C09149=1146.560,-113.783,-43.527,178.648,5.974,149.471
C09150=1146.565,-114.032,-43.519,178.646,5.974,149.471
C09151=1146.571,-114.282,-43.510,178.644,5.974,149.472
C09152=1146.576,-114.532,-43.501,178.642,5.973,149.472
C09153=1146.581,-114.781,-43.492,178.640,5.973,149.473
C09154=1146.587,-115.031,-43.484,178.638,5.973,149.473
C09155=1146.592,-115.281,-43.475,178.636,5.973,149.474
C09156=1146.598,-115.531,-43.466,178.634,5.972,149.474
C09157=1146.603,-115.781,-43.457,178.632,5.971,149.475
C09158=1146.609,-116.030,-43.449,178.630,5.971,149.475
C09159=1146.614,-116.280,-43.441,178.628,5.970,149.476
C09160=1146.619,-116.530,-43.432,178.627,5.970,149.476
C09161=1146.625,-116.779,-43.424,178.624,5.970,149.477
C09162=1146.630,-117.029,-43.415,178.622,5.970,149.477
C09163=1146.635,-117.279,-43.406,178.620,5.969,149.478
C09164=1146.641,-117.530,-43.398,178.619,5.969,149.478
C09165=1146.646,-117.779,-43.389,178.616,5.969,149.479
C09166=1146.651,-118.028,-43.380,178.614,5.968,149.479
C09167=1146.657,-118.278,-43.371,178.613,5.968,149.480
C09168=1146.663,-118.528,-43.363,178.610,5.967,149.480
C09169=1146.668,-118.778,-43.354,178.609,5.967,149.481
C09170=1146.673,-119.028,-43.346,178.607,5.967,149.481
C09171=1146.678,-119.278,-43.337,178.605,5.967,149.482
C09172=1146.684,-119.527,-43.329,178.602,5.966,149.482
C09173=1146.689,-119.777,-43.320,178.601,5.966,149.483
C09174=1146.695,-120.027,-43.311,178.599,5.966,149.483
C09175=1146.701,-120.277,-43.303,178.597,5.966,149.484
C09176=1146.706,-120.527,-43.294,178.595,5.965,149.484
C09177=1146.710,-120.776,-43.286,178.593,5.965,149.485
C09178=1146.716,-121.026,-43.278,178.591,5.964,149.485
C09179=1146.721,-121.276,-43.269,178.589,5.964,149.486
C09180=1146.727,-121.526,-43.260,178.587,5.963,149.486
C09181=1146.733,-121.776,-43.253,178.585,5.963,149.487
C09182=1146.738,-122.025,-43.244,178.583,5.963,149.487
C09183=1146.743,-122.275,-43.235,178.581,5.962,149.488
C09184=1146.749,-122.525,-43.227,178.579,5.962,149.489
C09185=1146.754,-122.775,-43.219,178.577,5.962,149.489
C09186=1146.759,-123.025,-43.211,178.575,5.962,149.490
C09187=1146.765,-123.274,-43.202,178.573,5.961,149.490
C09188=1146.770,-123.524,-43.193,178.571,5.961,149.491
C09189=1146.775,-123.775,-43.185,178.569,5.960,149.491
C09190=1146.781,-124.024,-43.176,178.568,5.960,149.491
C09191=1146.786,-124.273,-43.168,178.565,5.960,149.492
C09192=1146.791,-124.524,-43.160,178.564,5.960,149.492
C09193=1146.797,-124.773,-43.151,178.562,5.959,149.493
C09194=1146.802,-125.023,-43.143,178.560,5.959,149.493
C09195=1146.808,-125.273,-43.134,178.558,5.958,149.494
C09196=1146.814,-125.523,-43.126,178.556,5.958,149.494
C09197=1146.818,-125.772,-43.118,178.554,5.957,149.495
C09198=1146.824,-126.022,-43.110,178.553,5.957,149.495
C09199=1146.829,-126.272,-43.101,178.550,5.957,149.496
C09200=1146.834,-126.522,-43.093,178.548,5.957,149.497
C09201=1146.840,-126.772,-43.085,178.546,5.956,149.497
C09202=1146.845,-127.021,-43.076,178.544,5.956,149.498
C09203=1146.851,-127.271,-43.069,178.542,5.956,149.498
C09204=1146.856,-127.521,-43.060,178.541,5.956,149.499
C09205=1146.862,-127.771,-43.052,178.538,5.955,149.499
C09206=1146.867,-128.020,-43.043,178.537,5.955,149.500
C09207=1146.872,-128.271,-43.035,178.535,5.954,149.500
C09208=1146.452,-128.281,-43.078,178.531,5.958,149.502
C09209=1146.446,-128.032,-43.087,178.533,5.958,149.501
C09210=1146.441,-127.782,-43.094,178.535,5.959,149.501
C09211=1146.436,-127.532,-43.103,178.537,5.959,149.500
C09212=1146.430,-127.282,-43.111,178.539,5.959,149.500
C09213=1146.425,-127.033,-43.120,178.541,5.959,149.499
C09214=1146.419,-126.783,-43.128,178.543,5.960,149.499
C09215=1146.414,-126.533,-43.136,178.545,5.960,149.498
C09216=1146.409,-126.283,-43.144,178.547,5.961,149.498
C09217=1146.403,-126.034,-43.153,178.549,5.961,149.497
C09218=1146.397,-125.783,-43.161,178.551,5.961,149.497
C09219=1146.392,-125.534,-43.170,178.552,5.961,149.496
C09220=1146.387,-125.284,-43.177,178.555,5.962,149.496
C09221=1146.382,-125.034,-43.186,178.556,5.962,149.495
C09222=1146.376,-124.785,-43.195,178.558,5.963,149.495
C09223=1146.370,-124.534,-43.203,178.560,5.963,149.494
C09224=1146.365,-124.285,-43.212,178.562,5.964,149.494
C09225=1146.360,-124.035,-43.219,178.564,5.964,149.493
C09226=1146.355,-123.785,-43.228,178.566,5.964,149.493
C09227=1146.349,-123.536,-43.236,178.568,5.964,149.492
C09228=1146.344,-123.286,-43.244,178.570,5.965,149.492
C09229=1146.338,-123.036,-43.253,178.571,5.965,149.491
C09230=1146.332,-122.786,-43.261,178.574,5.965,149.491
C09231=1146.327,-122.536,-43.270,178.576,5.965,149.490
C09232=1146.323,-122.287,-43.278,178.578,5.966,149.490
C09233=1146.317,-122.037,-43.286,178.579,5.966,149.489
C09234=1146.311,-121.787,-43.295,178.582,5.967,149.489
C09235=1146.306,-121.537,-43.303,178.583,5.967,149.488
C09236=1146.300,-121.287,-43.312,178.585,5.967,149.488
C09237=1146.295,-121.038,-43.321,178.588,5.968,149.487
C09238=1146.290,-120.787,-43.329,178.589,5.968,149.487
C09239=1146.284,-120.538,-43.337,178.591,5.969,149.486
C09240=1146.279,-120.288,-43.346,178.593,5.969,149.486
C09241=1146.274,-120.039,-43.355,178.595,5.970,149.485
C09242=1146.269,-119.788,-43.363,178.597,5.969,149.485
C09243=1146.263,-119.539,-43.371,178.600,5.970,149.484
C09244=1146.258,-119.289,-43.380,178.601,5.970,149.484
C09245=1146.252,-119.039,-43.388,178.603,5.971,149.483
C09246=1146.247,-118.789,-43.397,178.605,5.971,149.483
C09247=1146.241,-118.540,-43.406,178.607,5.971,149.482
C09248=1146.236,-118.290,-43.415,178.609,5.971,149.482
C09249=1146.230,-118.040,-43.423,178.611,5.972,149.481
C09250=1146.225,-117.790,-43.431,178.613,5.972,149.481
C09251=1146.220,-117.540,-43.440,178.615,5.973,149.480
C09252=1146.214,-117.290,-43.449,178.617,5.973,149.480
C09253=1146.209,-117.041,-43.457,178.619,5.973,149.479
C09254=1146.203,-116.791,-43.466,178.621,5.974,149.478
C09255=1146.198,-116.541,-43.475,178.623,5.974,149.478
C09256=1146.193,-116.291,-43.484,178.625,5.975,149.478
C09257=1146.187,-116.041,-43.492,178.627,5.974,149.477
C09258=1146.182,-115.792,-43.500,178.629,5.975,149.477
C09259=1146.177,-115.542,-43.509,178.630,5.975,149.476
C09260=1146.171,-115.293,-43.518,178.633,5.976,149.476
C09261=1146.166,-115.043,-43.527,178.635,5.977,149.475
C09262=1146.160,-114.792,-43.535,178.637,5.976,149.474
C09263=1146.155,-114.542,-43.544,178.639,5.977,149.474
C09264=1146.149,-114.293,-43.552,178.641,5.977,149.473
C09265=1146.144,-114.043,-43.561,178.643,5.978,149.473
C09266=1146.139,-113.793,-43.570,178.644,5.978,149.472
C09267=1146.134,-113.544,-43.579,178.647,5.978,149.472
C09268=1146.128,-113.294,-43.587,178.648,5.978,149.471
C09269=1146.123,-113.044,-43.596,178.650,5.979,149.471
C09270=1146.117,-112.794,-43.605,178.653,5.980,149.470
C09271=1146.112,-112.544,-43.614,178.655,5.979,149.470
C09272=1146.107,-112.294,-43.623,178.657,5.980,149.469
C09273=1146.101,-112.045,-43.631,178.658,5.980,149.469
C09274=1146.096,-111.795,-43.640,178.661,5.981,149.468
C09275=1146.091,-111.546,-43.649,178.662,5.981,149.468
C09276=1146.086,-111.295,-43.657,178.664,5.982,149.467
C09277=1146.080,-111.045,-43.666,178.667,5.982,149.467
C09278=1146.075,-110.796,-43.674,178.669,5.982,149.466
C09279=1146.069,-110.546,-43.683,178.671,5.983,149.466
C09280=1146.064,-110.296,-43.693,178.673,5.983,149.465
C09281=1146.058,-110.046,-43.702,178.675,5.983,149.465
C09282=1146.053,-109.796,-43.711,178.676,5.983,149.464
C09283=1146.047,-109.547,-43.719,178.679,5.984,149.464
C09284=1146.042,-109.297,-43.728,178.681,5.985,149.463
C09285=1146.037,-109.048,-43.737,178.682,5.985,149.463
C09286=1146.032,-108.798,-43.746,178.685,5.985,149.462
C09287=1146.027,-108.548,-43.755,178.687,5.985,149.462
C09288=1146.022,-108.298,-43.764,178.689,5.986,149.461
C09289=1146.015,-108.049,-43.773,178.691,5.987,149.461
C09290=1146.010,-107.799,-43.782,178.693,5.987,149.460
C09291=1146.005,-107.549,-43.791,178.695,5.987,149.460
C09292=1146.000,-107.299,-43.799,178.697,5.987,149.459
C09293=1145.994,-107.049,-43.808,178.699,5.988,149.458
C09294=1145.989,-106.799,-43.817,178.701,5.988,149.458
C09295=1145.984,-106.550,-43.826,178.703,5.988,149.457
C09296=1145.978,-106.300,-43.835,178.705,5.989,149.457
C09297=1145.972,-106.050,-43.844,178.707,5.989,149.456
C09298=1145.967,-105.800,-43.853,178.709,5.990,149.456
C09299=1145.962,-105.550,-43.862,178.711,5.989,149.455
C09300=1145.957,-105.301,-43.871,178.713,5.990,149.455
C09301=1145.952,-105.051,-43.880,178.715,5.991,149.454
C09302=1145.946,-104.801,-43.889,178.717,5.991,149.454
C09303=1145.940,-104.551,-43.898,178.719,5.992,149.453
C09304=1145.935,-104.302,-43.907,178.721,5.992,149.453
C09305=1145.930,-104.052,-43.916,178.723,5.992,149.452
C09306=1145.925,-103.802,-43.925,178.726,5.993,149.452
C09307=1145.919,-103.552,-43.935,178.727,5.993,149.451
C09308=1145.914,-103.302,-43.944,178.729,5.993,149.451
C09309=1145.908,-103.030,-43.953,178.732,5.994,149.450
C09310=1145.903,-102.758,-43.963,178.734,5.994,149.449
C09311=1145.896,-102.487,-43.973,178.736,5.995,149.449
C09312=1145.891,-102.214,-43.983,178.739,5.995,149.448
C09313=1145.886,-101.964,-43.992,178.741,5.996,149.448
C09314=1145.880,-101.714,-44.001,178.742,5.996,149.447
C09315=1145.875,-101.465,-44.011,178.745,5.996,149.447
C09316=1145.870,-101.215,-44.020,178.746,5.996,149.446
C09317=1145.864,-100.965,-44.029,178.749,5.997,149.446
C09318=1145.859,-100.715,-44.038,178.751,5.997,149.445
C09319=1145.853,-100.465,-44.047,178.753,5.997,149.445
C09320=1145.848,-100.215,-44.056,178.755,5.998,149.444
C09321=1145.843,-99.966,-44.066,178.756,5.998,149.444
C09322=1145.837,-99.716,-44.075,178.759,5.999,149.443
C09323=1145.832,-99.466,-44.084,178.761,5.999,149.442
C09324=1145.827,-99.216,-44.093,178.763,5.999,149.442
C09325=1145.821,-98.967,-44.103,178.765,6.000,149.441
C09326=1145.816,-98.718,-44.111,178.767,6.001,149.441
C09327=1145.811,-98.468,-44.120,178.769,6.001,149.441
C09328=1145.805,-98.218,-44.130,178.771,6.001,149.440
C09329=1145.799,-97.968,-44.139,178.773,6.001,149.439
C09330=1145.795,-97.719,-44.148,178.775,6.002,149.439
C09331=1145.789,-97.468,-44.158,178.777,6.003,149.438
C09332=1145.784,-97.219,-44.167,178.779,6.003,149.438
C09333=1145.779,-96.969,-44.176,178.782,6.003,149.437
C09334=1145.773,-96.719,-44.186,178.784,6.004,149.437
C09335=1145.768,-96.469,-44.195,178.786,6.004,149.436
C09336=1145.762,-96.219,-44.204,178.788,6.004,149.436
C09337=1145.757,-95.970,-44.214,178.790,6.005,149.435
C09338=1145.752,-95.720,-44.223,178.792,6.005,149.434
C09339=1145.746,-95.470,-44.232,178.794,6.005,149.434
C09340=1145.741,-95.221,-44.242,178.796,6.006,149.434
C09341=1145.736,-94.971,-44.251,178.798,6.006,149.433
C09342=1145.730,-94.721,-44.260,178.800,6.007,149.433
C09343=1145.725,-94.471,-44.270,178.802,6.007,149.432
C09344=1145.719,-94.221,-44.279,178.804,6.007,149.431
C09345=1145.714,-93.971,-44.288,178.807,6.008,149.431
C09346=1145.709,-93.722,-44.298,178.808,6.008,149.430
C09347=1145.703,-93.472,-44.307,178.811,6.008,149.430
C09348=1145.698,-93.223,-44.317,178.813,6.009,149.429
C09349=1145.692,-92.973,-44.326,178.815,6.009,149.429
C09350=1145.687,-92.723,-44.335,178.817,6.010,149.428
C09351=1145.682,-92.474,-44.345,178.819,6.011,149.428
C09352=1145.676,-92.223,-44.354,178.821,6.010,149.427
C09353=1145.672,-91.974,-44.364,178.823,6.011,149.427
C09354=1145.666,-91.723,-44.374,178.826,6.012,149.426
C09355=1145.661,-91.473,-44.383,178.827,6.012,149.426
C09356=1145.656,-91.224,-44.393,178.830,6.012,149.425
C09357=1145.650,-90.974,-44.402,178.832,6.013,149.424
C09358=1145.645,-90.724,-44.412,178.834,6.013,149.424
C09359=1145.640,-90.475,-44.421,178.836,6.014,149.423
C09360=1145.635,-90.225,-44.431,178.838,6.014,149.423
C09361=1145.629,-89.975,-44.440,178.840,6.014,149.422
C09362=1145.624,-89.726,-44.450,178.842,6.015,149.422
C09363=1145.618,-89.476,-44.459,178.844,6.015,149.421
C09364=1145.613,-89.227,-44.469,178.846,6.015,149.421
C09365=1145.607,-88.976,-44.478,178.849,6.016,149.420
C09366=1145.602,-88.727,-44.488,178.851,6.017,149.420
C09367=1145.597,-88.477,-44.498,178.852,6.017,149.419
C09368=1145.592,-88.227,-44.507,178.855,6.017,149.419
C09369=1145.586,-87.977,-44.517,178.857,6.018,149.418
C09370=1145.582,-87.728,-44.527,178.859,6.018,149.417
C09371=1145.576,-87.478,-44.536,178.861,6.018,149.417
C09372=1145.571,-87.228,-44.546,178.863,6.019,149.416
C09373=1145.565,-86.978,-44.555,178.866,6.020,149.416
C09374=1145.560,-86.729,-44.565,178.868,6.019,149.415
C09375=1145.554,-86.479,-44.574,178.870,6.020,149.415
C09376=1145.549,-86.228,-44.585,178.872,6.021,149.414
C09377=1145.544,-85.979,-44.594,178.874,6.021,149.414
C09378=1145.538,-85.729,-44.604,178.876,6.021,149.413
C09379=1145.533,-85.480,-44.614,178.878,6.022,149.413
C09380=1145.528,-85.230,-44.623,178.880,6.022,149.412
C09381=1145.523,-84.980,-44.633,178.883,6.022,149.411
C09382=1145.517,-84.731,-44.643,178.885,6.023,149.411
C09383=1145.513,-84.480,-44.652,178.887,6.023,149.410
C09384=1145.507,-84.231,-44.662,178.889,6.024,149.410
C09385=1145.501,-83.981,-44.672,178.891,6.024,149.409
C09386=1145.496,-83.731,-44.681,178.894,6.025,149.409
C09387=1145.491,-83.482,-44.692,178.895,6.025,149.408
C09388=1145.485,-83.232,-44.701,178.897,6.026,149.408
C09389=1145.480,-82.983,-44.711,178.900,6.026,149.407
C09390=1145.475,-82.732,-44.721,178.902,6.026,149.407
C09391=1145.470,-82.482,-44.730,178.904,6.027,149.406
C09392=1145.464,-82.233,-44.740,178.906,6.028,149.406
C09393=1145.458,-81.983,-44.751,178.908,6.027,149.405
C09394=1145.453,-81.733,-44.760,178.910,6.028,149.404
C09395=1145.448,-81.483,-44.770,178.912,6.029,149.404
C09396=1145.443,-81.234,-44.780,178.915,6.030,149.403
C09397=1145.438,-80.984,-44.790,178.917,6.029,149.403
C09398=1145.432,-80.734,-44.799,178.919,6.030,149.402
C09399=1145.426,-80.485,-44.810,178.921,6.031,149.402
C09400=1145.422,-80.235,-44.820,178.923,6.031,149.401
C09401=1145.416,-79.985,-44.829,178.925,6.031,149.401
C09402=1145.411,-79.735,-44.839,178.928,6.032,149.400
C09403=1145.406,-79.486,-44.849,178.930,6.033,149.400
C09404=1145.400,-79.236,-44.859,178.932,6.032,149.399
C09405=1145.395,-78.986,-44.870,178.934,6.033,149.398
C09406=1145.390,-78.736,-44.879,178.936,6.034,149.398
C09407=1145.384,-78.487,-44.889,178.938,6.034,149.397
C09408=1145.379,-78.237,-44.899,178.941,6.034,149.397
C09409=1145.373,-77.988,-44.909,178.943,6.035,149.396
C09410=1145.369,-77.737,-44.919,178.945,6.036,149.396
C09411=1145.363,-77.488,-44.929,178.947,6.035,149.395
C09412=1145.357,-77.238,-44.939,178.949,6.036,149.395
C09413=1145.352,-76.967,-44.950,178.951,6.037,149.394
C09414=1145.346,-76.695,-44.961,178.954,6.037,149.393
C09415=1145.340,-76.424,-44.971,178.956,6.038,149.393
C09416=1145.334,-76.152,-44.983,178.959,6.038,149.392
C09417=1145.329,-75.903,-44.992,178.961,6.039,149.392
C09418=1145.324,-75.653,-45.003,178.963,6.039,149.391
C09419=1145.319,-75.403,-45.013,178.965,6.039,149.391
C09420=1145.313,-75.153,-45.023,178.968,6.040,149.390
C09421=1145.308,-74.904,-45.032,178.970,6.041,149.390
C09422=1145.303,-74.654,-45.043,178.971,6.041,149.389
C09423=1145.297,-74.404,-45.053,178.974,6.041,149.388
C09424=1145.292,-74.154,-45.063,178.976,6.042,149.388
C09425=1145.286,-73.905,-45.074,178.978,6.043,149.387
C09426=1145.282,-73.655,-45.084,178.980,6.042,149.387
C09427=1145.276,-73.405,-45.094,178.983,6.043,149.386
C09428=1145.271,-73.156,-45.104,178.985,6.044,149.386
C09429=1145.266,-72.906,-45.115,178.987,6.045,149.385
C09430=1145.260,-72.656,-45.125,178.989,6.044,149.385
C09431=1145.255,-72.407,-45.135,178.991,6.045,149.384
C09432=1145.250,-72.157,-45.145,178.994,6.046,149.384
C09433=1145.244,-71.906,-45.154,178.996,6.046,149.383
C09434=1145.239,-71.657,-45.165,178.998,6.046,149.382
C09435=1145.233,-71.407,-45.175,179.000,6.047,149.382
C09436=1145.228,-71.157,-45.185,179.003,6.047,149.381
C09437=1145.223,-70.908,-45.196,179.005,6.048,149.381
C09438=1145.217,-70.658,-45.206,179.006,6.048,149.380
C09439=1145.213,-70.408,-45.216,179.009,6.048,149.380
C09440=1145.207,-70.159,-45.226,179.011,6.049,149.379
C09441=1145.202,-69.910,-45.237,179.013,6.050,149.379
C09442=1145.197,-69.659,-45.248,179.015,6.050,149.378
C09443=1145.191,-69.410,-45.258,179.018,6.050,149.377
C09444=1145.186,-69.160,-45.268,179.020,6.051,149.377
C09445=1145.181,-68.910,-45.278,179.022,6.052,149.376
C09446=1145.175,-68.661,-45.289,179.025,6.052,149.376
C09447=1145.170,-68.410,-45.299,179.026,6.052,149.375
C09448=1145.164,-68.161,-45.309,179.029,6.053,149.375
C09449=1145.160,-67.912,-45.319,179.031,6.053,149.374
C09450=1145.155,-67.661,-45.330,179.033,6.054,149.374
C09451=1145.149,-67.412,-45.340,179.036,6.055,149.373
C09452=1145.143,-67.162,-45.350,179.038,6.054,149.372
C09453=1145.138,-66.912,-45.361,179.040,6.055,149.372
C09454=1145.133,-66.663,-45.372,179.042,6.056,149.371
C09455=1145.128,-66.413,-45.382,179.044,6.057,149.371
C09456=1145.123,-66.163,-45.392,179.046,6.056,149.370
C09457=1145.117,-65.914,-45.403,179.049,6.057,149.370
C09458=1145.112,-65.663,-45.413,179.051,6.058,149.369
C09459=1145.106,-65.414,-45.423,179.053,6.058,149.369
C09460=1145.101,-65.164,-45.434,179.056,6.059,149.368
C09461=1145.096,-64.915,-45.445,179.057,6.059,149.368
C09462=1145.091,-64.665,-45.455,179.060,6.059,149.367
C09463=1145.085,-64.415,-45.466,179.062,6.060,149.366
C09464=1145.080,-64.165,-45.476,179.064,6.061,149.366
C09465=1145.075,-63.915,-45.486,179.067,6.061,149.365
C09466=1145.070,-63.666,-45.497,179.068,6.061,149.365
C09467=1145.065,-63.416,-45.508,179.071,6.062,149.364
C09468=1145.059,-63.166,-45.518,179.073,6.063,149.364
C09469=1145.054,-62.916,-45.529,179.076,6.063,149.363
C09470=1145.048,-62.667,-45.539,179.078,6.064,149.363
C09471=1145.043,-62.418,-45.550,179.080,6.064,149.362
C09472=1145.038,-62.168,-45.560,179.082,6.064,149.361
C09473=1145.032,-61.918,-45.571,179.084,6.065,149.361
C09474=1145.027,-61.668,-45.581,179.087,6.066,149.360
C09475=1145.022,-61.419,-45.592,179.089,6.066,149.360
C09476=1145.017,-61.169,-45.603,179.091,6.067,149.359
C09477=1145.012,-60.919,-45.613,179.093,6.067,149.359
C09478=1145.007,-60.669,-45.624,179.095,6.068,149.358
C09479=1145.001,-60.420,-45.634,179.098,6.068,149.358
C09480=1144.996,-60.170,-45.645,179.100,6.069,149.357
C09481=1144.990,-59.920,-45.657,179.103,6.069,149.356
C09482=1144.985,-59.670,-45.667,179.105,6.070,149.356
C09483=1144.980,-59.421,-45.677,179.107,6.070,149.355
C09484=1144.975,-59.171,-45.689,179.109,6.071,149.355
C09485=1144.969,-58.921,-45.699,179.111,6.071,149.354
C09486=1144.964,-58.671,-45.709,179.114,6.072,149.354
C09487=1144.959,-58.422,-45.720,179.116,6.073,149.353
C09488=1144.954,-58.172,-45.731,179.118,6.073,149.353
C09489=1144.949,-57.922,-45.741,179.120,6.073,149.352
C09490=1144.943,-57.673,-45.753,179.122,6.074,149.351
C09491=1144.937,-57.423,-45.763,179.125,6.074,149.351
C09492=1144.933,-57.173,-45.774,179.127,6.075,149.350
C09493=1144.927,-56.924,-45.785,179.130,6.076,149.350
C09494=1144.922,-56.674,-45.795,179.132,6.076,149.349
C09495=1144.918,-56.424,-45.807,179.134,6.076,149.349
C09496=1144.912,-56.174,-45.817,179.136,6.077,149.348
C09497=1144.906,-55.924,-45.829,179.138,6.078,149.348
C09498=1144.901,-55.675,-45.839,179.141,6.078,149.347
C09499=1144.896,-55.425,-45.850,179.143,6.079,149.346
C09500=1144.891,-55.176,-45.860,179.145,6.080,149.346
C09501=1144.886,-54.926,-45.872,179.148,6.080,149.345
C09502=1144.880,-54.677,-45.882,179.149,6.080,149.345
C09503=1144.875,-54.427,-45.894,179.152,6.080,149.344
C09504=1144.870,-54.176,-45.904,179.154,6.081,149.344
C09505=1144.865,-53.927,-45.915,179.157,6.082,149.343
C09506=1144.860,-53.677,-45.926,179.159,6.082,149.342
C09507=1144.854,-53.428,-45.937,179.161,6.083,149.342
C09508=1144.849,-53.178,-45.948,179.164,6.084,149.341
C09509=1144.844,-52.928,-45.959,179.166,6.083,149.341
C09510=1144.838,-52.679,-45.969,179.168,6.084,149.340
C09511=1144.834,-52.429,-45.981,179.170,6.085,149.340
C09512=1144.827,-52.179,-45.991,179.173,6.085,149.339
C09513=1144.823,-51.929,-46.003,179.175,6.086,149.339
C09514=1144.818,-51.679,-46.013,179.177,6.087,149.338
C09515=1144.812,-51.430,-46.024,179.180,6.087,149.337
C09516=1144.807,-51.180,-46.035,179.181,6.087,149.337
C09517=1144.800,-50.909,-46.047,179.185,6.088,149.336
C09518=1144.795,-50.639,-46.059,179.187,6.089,149.336
C09519=1144.790,-50.368,-46.071,179.189,6.090,149.335
C09520=1144.784,-50.098,-46.083,179.192,6.090,149.335
C09521=1144.779,-49.848,-46.094,179.194,6.091,149.334
C09522=1144.773,-49.598,-46.106,179.196,6.091,149.333
C09523=1144.768,-49.348,-46.116,179.198,6.092,149.333
C09524=1144.763,-49.099,-46.128,179.201,6.092,149.332
C09525=1144.757,-48.848,-46.139,179.203,6.093,149.332
C09526=1144.752,-48.599,-46.150,179.206,6.093,149.331
C09527=1144.747,-48.350,-46.161,179.208,6.094,149.331
C09528=1144.741,-48.100,-46.172,179.210,6.095,149.330
C09529=1144.736,-47.850,-46.183,179.213,6.095,149.329
C09530=1144.732,-47.601,-46.195,179.215,6.096,149.329
C09531=1144.726,-47.351,-46.206,179.216,6.096,149.328
C09532=1144.721,-47.101,-46.217,179.219,6.096,149.328
C09533=1144.716,-46.851,-46.228,179.221,6.097,149.327
C09534=1144.711,-46.602,-46.240,179.223,6.098,149.327
C09535=1144.705,-46.352,-46.250,179.226,6.098,149.326
C09536=1144.700,-46.102,-46.261,179.228,6.099,149.326
C09537=1144.695,-45.852,-46.273,179.231,6.099,149.325
C09538=1144.690,-45.604,-46.284,179.233,6.100,149.324
C09539=1144.684,-45.353,-46.295,179.235,6.101,149.324
C09540=1144.679,-45.103,-46.307,179.238,6.101,149.323
C09541=1144.673,-44.854,-46.318,179.240,6.101,149.323
C09542=1144.668,-44.604,-46.329,179.242,6.102,149.322
C09543=1144.663,-44.354,-46.340,179.244,6.103,149.322
C09544=1144.658,-44.104,-46.352,179.247,6.103,149.321
C09545=1144.653,-43.855,-46.363,179.249,6.104,149.320
C09546=1144.647,-43.605,-46.375,179.252,6.105,149.320
C09547=1144.643,-43.356,-46.386,179.254,6.105,149.319
C09548=1144.637,-43.107,-46.397,179.256,6.106,149.319
C09549=1144.632,-42.856,-46.408,179.259,6.106,149.318
C09550=1144.627,-42.607,-46.419,179.261,6.107,149.318
C09551=1144.621,-42.357,-46.431,179.263,6.108,149.317
C09552=1144.616,-42.108,-46.442,179.266,6.108,149.317
C09553=1144.611,-41.858,-46.454,179.268,6.108,149.316
C09554=1144.606,-41.608,-46.465,179.270,6.109,149.315
C09555=1144.601,-41.358,-46.477,179.272,6.110,149.315
C09556=1144.595,-41.109,-46.487,179.275,6.110,149.314
C09557=1144.590,-40.859,-46.499,179.277,6.111,149.314
C09558=1144.585,-40.609,-46.511,179.279,6.112,149.313
C09559=1144.579,-40.359,-46.522,179.282,6.112,149.313
C09560=1144.575,-40.110,-46.534,179.284,6.113,149.312
C09561=1144.569,-39.860,-46.545,179.287,6.113,149.311
C09562=1144.564,-39.611,-46.557,179.289,6.114,149.311
C09563=1144.559,-39.361,-46.568,179.291,6.115,149.311
C09564=1144.553,-39.111,-46.580,179.294,6.115,149.310
C09565=1144.548,-38.862,-46.591,179.296,6.116,149.309
C09566=1144.542,-38.612,-46.603,179.298,6.116,149.309
C09567=1144.538,-38.362,-46.614,179.301,6.117,149.308
C09568=1144.532,-38.113,-46.626,179.303,6.118,149.308
C09569=1144.528,-37.863,-46.638,179.306,6.118,149.307
C09570=1144.522,-37.614,-46.649,179.307,6.118,149.307
C09571=1144.516,-37.364,-46.661,179.309,6.119,149.306
C09572=1144.511,-37.114,-46.672,179.312,6.120,149.305
C09573=1144.506,-36.864,-46.684,179.314,6.120,149.305
C09574=1144.501,-36.615,-46.695,179.317,6.121,149.304
C09575=1144.496,-36.365,-46.707,179.319,6.121,149.304
C09576=1144.490,-36.115,-46.719,179.321,6.122,149.303
C09577=1144.485,-35.866,-46.730,179.324,6.123,149.302
C09578=1144.480,-35.616,-46.742,179.326,6.123,149.302
C09579=1144.475,-35.366,-46.753,179.329,6.124,149.301
C09580=1144.470,-35.116,-46.765,179.331,6.125,149.301
C09581=1144.464,-34.866,-46.777,179.333,6.125,149.300
C09582=1144.460,-34.617,-46.788,179.336,6.126,149.300
C09583=1144.454,-34.367,-46.800,179.338,6.127,149.299
C09584=1144.448,-34.117,-46.812,179.341,6.127,149.299
C09585=1144.443,-33.868,-46.823,179.343,6.128,149.298
C09586=1144.438,-33.619,-46.836,179.345,6.129,149.298
C09587=1144.433,-33.369,-46.848,179.348,6.129,149.297
C09588=1144.428,-33.119,-46.859,179.350,6.130,149.296
C09589=1144.423,-32.869,-46.871,179.352,6.131,149.296
C09590=1144.417,-32.619,-46.883,179.355,6.131,149.295
C09591=1144.412,-32.370,-46.894,179.357,6.132,149.295
C09592=1144.407,-32.120,-46.905,179.359,6.132,149.294
C09593=1144.401,-31.871,-46.918,179.362,6.133,149.294
C09594=1144.397,-31.621,-46.929,179.364,6.134,149.293
C09595=1144.391,-31.371,-46.941,179.367,6.134,149.292
C09596=1144.386,-31.121,-46.953,179.369,6.135,149.292
C09597=1144.380,-30.872,-46.965,179.371,6.135,149.291
C09598=1144.376,-30.623,-46.977,179.374,6.136,149.291
C09599=1144.371,-30.373,-46.989,179.376,6.137,149.290
C09600=1144.365,-30.123,-47.001,179.378,6.137,149.290
C09601=1144.360,-29.873,-47.013,179.381,6.138,149.289
C09602=1144.355,-29.624,-47.025,179.383,6.139,149.288
C09603=1144.349,-29.374,-47.036,179.385,6.139,149.288
C09604=1144.344,-29.125,-47.048,179.388,6.140,149.287
C09605=1144.339,-28.875,-47.060,179.390,6.141,149.287
C09606=1144.334,-28.626,-47.072,179.392,6.141,149.286
C09607=1144.329,-28.376,-47.084,179.395,6.142,149.286
C09608=1144.323,-28.126,-47.096,179.397,6.143,149.285
C09609=1144.318,-27.876,-47.108,179.399,6.143,149.285
C09610=1144.313,-27.627,-47.120,179.402,6.144,149.284
C09611=1144.308,-27.377,-47.132,179.404,6.145,149.283
C09612=1144.303,-27.128,-47.144,179.407,6.145,149.283
C09613=1144.297,-26.878,-47.156,179.409,6.146,149.282
C09614=1144.292,-26.628,-47.168,179.411,6.147,149.282
C09615=1144.287,-26.378,-47.180,179.414,6.147,149.281
C09616=1144.282,-26.129,-47.192,179.416,6.148,149.281
C09617=1144.277,-25.879,-47.204,179.419,6.148,149.280
C09618=1144.272,-25.629,-47.216,179.421,6.149,149.279
C09619=1144.266,-25.379,-47.228,179.423,6.150,149.279
C09620=1144.261,-25.130,-47.240,179.426,6.150,149.278
C09621=1144.256,-24.860,-47.254,179.428,6.151,149.278
C09622=1144.250,-24.590,-47.266,179.431,6.151,149.277
C09623=1144.245,-24.320,-47.279,179.433,6.152,149.276
C09624=1144.239,-24.049,-47.293,179.436,6.153,149.276
C09625=1144.234,-23.800,-47.305,179.439,6.154,149.275
C09626=1144.229,-23.550,-47.317,179.441,6.155,149.275
C09627=1144.224,-23.301,-47.329,179.443,6.155,149.274
C09628=1144.218,-23.051,-47.341,179.446,6.156,149.274
C09629=1144.213,-22.802,-47.354,179.448,6.157,149.273
C09630=1144.208,-22.552,-47.366,179.451,6.157,149.272
C09631=1144.202,-22.302,-47.378,179.453,6.158,149.272
C09632=1144.197,-22.052,-47.390,179.455,6.159,149.272
C09633=1144.192,-21.803,-47.402,179.458,6.159,149.271
C09634=1144.187,-21.553,-47.415,179.460,6.160,149.270
C09635=1144.181,-21.303,-47.427,179.463,6.160,149.270
C09636=1144.176,-21.054,-47.439,179.465,6.161,149.269
C09637=1144.171,-20.805,-47.452,179.467,6.162,149.269
C09638=1144.165,-20.555,-47.464,179.470,6.162,149.268
C09639=1144.160,-20.305,-47.476,179.472,6.163,149.268
C09640=1144.155,-20.055,-47.488,179.474,6.163,149.267
C09641=1144.150,-19.805,-47.501,179.477,6.164,149.266
C09642=1144.146,-19.556,-47.512,179.480,6.165,149.266
C09643=1144.141,-19.306,-47.525,179.482,6.166,149.265
C09644=1144.135,-19.057,-47.538,179.484,6.167,149.265
C09645=1144.130,-18.807,-47.549,179.487,6.167,149.264
C09646=1144.124,-18.558,-47.563,179.489,6.168,149.264
C09647=1144.119,-18.308,-47.575,179.492,6.169,149.263
C09648=1144.114,-18.058,-47.587,179.494,6.169,149.262
C09649=1144.108,-17.809,-47.600,179.496,6.170,149.262
C09650=1144.104,-17.558,-47.612,179.499,6.171,149.261
C09651=1144.098,-17.309,-47.625,179.501,6.171,149.261
C09652=1144.093,-17.060,-47.637,179.504,6.172,149.260
C09653=1144.088,-16.810,-47.649,179.506,6.173,149.260
C09654=1144.083,-16.560,-47.662,179.508,6.174,149.259
C09655=1144.078,-16.311,-47.674,179.511,6.174,149.258
C09656=1144.072,-16.061,-47.686,179.513,6.176,149.258
C09657=1144.068,-15.811,-47.699,179.516,6.176,149.257
C09658=1144.063,-15.562,-47.712,179.518,6.177,149.257
C09659=1144.057,-15.312,-47.724,179.521,6.177,149.256
C09660=1144.052,-15.063,-47.736,179.523,6.178,149.256
C09661=1144.047,-14.813,-47.749,179.525,6.179,149.255
C09662=1144.042,-14.564,-47.761,179.528,6.179,149.255
C09663=1144.036,-14.313,-47.774,179.530,6.180,149.254
C09664=1144.031,-14.064,-47.787,179.533,6.180,149.253
C09665=1144.026,-13.814,-47.799,179.535,6.181,149.253
C09666=1144.021,-13.565,-47.812,179.537,6.182,149.252
C09667=1144.015,-13.315,-47.824,179.540,6.183,149.252
C09668=1144.010,-13.066,-47.837,179.543,6.184,149.251
C09669=1144.006,-12.816,-47.850,179.545,6.184,149.251
C09670=1144.001,-12.567,-47.862,179.547,6.185,149.250
C09671=1143.995,-12.317,-47.875,179.550,6.186,149.250
C09672=1143.989,-12.067,-47.887,179.552,6.186,149.249
C09673=1143.985,-11.817,-47.900,179.554,6.187,149.248
C09674=1143.980,-11.568,-47.913,179.557,6.188,149.248
C09675=1143.975,-11.318,-47.925,179.559,6.188,149.247
C09676=1143.969,-11.069,-47.938,179.562,6.189,149.247
C09677=1143.964,-10.819,-47.951,179.565,6.191,149.246
C09678=1143.959,-10.569,-47.963,179.567,6.191,149.246
C09679=1143.954,-10.319,-47.976,179.570,6.192,149.245
C09680=1143.949,-10.070,-47.989,179.572,6.193,149.244
C09681=1143.943,-9.821,-48.001,179.574,6.193,149.244
C09682=1143.938,-9.570,-48.015,179.577,6.194,149.243
C09683=1143.933,-9.321,-48.027,179.579,6.195,149.243
C09684=1143.928,-9.072,-48.040,179.581,6.195,149.242
C09685=1143.923,-8.822,-48.053,179.584,6.197,149.242
C09686=1143.918,-8.572,-48.066,179.587,6.197,149.241
C09687=1143.912,-8.323,-48.079,179.589,6.198,149.241
C09688=1143.907,-8.074,-48.091,179.591,6.199,149.240
C09689=1143.903,-7.824,-48.104,179.594,6.199,149.239
C09690=1143.897,-7.574,-48.118,179.596,6.200,149.239
C09691=1143.892,-7.325,-48.130,179.599,6.200,149.238
C09692=1143.887,-7.075,-48.143,179.601,6.201,149.238
C09693=1143.882,-6.825,-48.156,179.604,6.202,149.237
C09694=1143.876,-6.576,-48.169,179.606,6.203,149.237
C09695=1143.871,-6.326,-48.181,179.608,6.204,149.236
C09696=1143.867,-6.076,-48.194,179.611,6.204,149.235
C09697=1143.861,-5.827,-48.208,179.613,6.205,149.235
C09698=1143.856,-5.577,-48.220,179.616,6.206,149.234
C09699=1143.851,-5.327,-48.233,179.618,6.206,149.234
C09700=1143.845,-5.078,-48.246,179.621,6.208,149.233
C09701=1143.840,-4.828,-48.259,179.624,6.208,149.233
C09702=1143.836,-4.578,-48.272,179.626,6.209,149.232
C09703=1143.830,-4.329,-48.285,179.628,6.210,149.232
C09704=1143.825,-4.079,-48.298,179.631,6.210,149.231
C09705=1143.820,-3.829,-48.311,179.633,6.211,149.230
C09706=1143.814,-3.580,-48.324,179.636,6.212,149.230
C09707=1143.809,-3.330,-48.337,179.638,6.213,149.229
C09708=1143.805,-3.081,-48.350,179.641,6.214,149.229
C09709=1143.799,-2.831,-48.363,179.643,6.215,149.228
C09710=1143.794,-2.582,-48.376,179.646,6.215,149.228
C09711=1143.789,-2.332,-48.390,179.648,6.216,149.227
C09712=1143.784,-2.082,-48.402,179.651,6.217,149.227
C09713=1143.778,-1.833,-48.415,179.653,6.218,149.226
C09714=1143.773,-1.583,-48.428,179.655,6.219,149.225
C09715=1143.768,-1.334,-48.442,179.658,6.219,149.225
C09716=1143.763,-1.084,-48.455,179.660,6.220,149.224
C09717=1143.758,-0.834,-48.468,179.663,6.220,149.224
C09718=1143.753,-0.585,-48.480,179.666,6.222,149.223
C09719=1143.748,-0.335,-48.495,179.668,6.223,149.223
C09720=1143.743,-0.086,-48.507,179.671,6.223,149.222
C09721=1143.737,0.164,-48.521,179.673,6.224,149.222
C09722=1143.732,0.414,-48.533,179.675,6.224,149.221
C09723=1143.726,0.663,-48.547,179.678,6.225,149.220
C09724=1143.722,0.913,-48.560,179.680,6.227,149.220
C09725=1143.717,1.183,-48.575,179.683,6.227,149.219
C09726=1143.710,1.451,-48.589,179.686,6.228,149.219
C09727=1143.705,1.721,-48.603,179.688,6.229,149.218
C09728=1143.700,1.990,-48.618,179.691,6.230,149.217
C09729=1143.695,2.240,-48.631,179.693,6.230,149.217
C09730=1143.690,2.490,-48.644,179.697,6.232,149.216
C09731=1143.684,2.740,-48.657,179.699,6.233,149.216
C09732=1143.679,2.988,-48.671,179.701,6.233,149.215
C09733=1143.674,3.239,-48.684,179.704,6.234,149.215
C09734=1143.669,3.487,-48.697,179.706,6.235,149.214
C09735=1143.664,3.738,-48.711,179.709,6.236,149.213
C09736=1143.659,3.987,-48.724,179.711,6.237,149.213
C09737=1143.654,4.237,-48.738,179.714,6.237,149.212
C09738=1143.648,4.486,-48.751,179.716,6.238,149.212
C09739=1143.643,4.737,-48.764,179.718,6.239,149.211
C09740=1143.638,4.985,-48.777,179.721,6.240,149.211
C09741=1143.633,5.236,-48.791,179.724,6.241,149.210
C09742=1143.628,5.485,-48.805,179.726,6.241,149.210
C09743=1143.623,5.735,-48.818,179.728,6.242,149.209
C09744=1143.617,5.984,-48.832,179.731,6.243,149.209
C09745=1143.613,6.234,-48.845,179.734,6.244,149.208
C09746=1143.607,6.483,-48.858,179.736,6.245,149.208
C09747=1143.602,6.733,-48.872,179.739,6.245,149.207
C09748=1143.597,6.982,-48.885,179.741,6.246,149.206
C09749=1143.592,7.232,-48.899,179.744,6.247,149.206
C09750=1143.587,7.481,-48.912,179.746,6.248,149.205
C09751=1143.582,7.731,-48.926,179.748,6.249,149.205
C09752=1143.576,7.981,-48.939,179.751,6.249,149.204
C09753=1143.572,8.230,-48.953,179.754,6.251,149.204
C09754=1143.567,8.480,-48.966,179.757,6.251,149.203
C09755=1143.561,8.729,-48.980,179.759,6.252,149.202
C09756=1143.557,8.979,-48.993,179.761,6.253,149.202
C09757=1143.551,9.228,-49.007,179.764,6.253,149.201
C09758=1143.546,9.478,-49.021,179.766,6.255,149.201
C09759=1143.541,9.727,-49.034,179.769,6.256,149.200
C09760=1143.536,9.977,-49.048,179.771,6.256,149.200
C09761=1143.530,10.227,-49.062,179.773,6.257,149.199
C09762=1143.525,10.476,-49.076,179.777,6.258,149.199
C09763=1143.521,10.726,-49.089,179.779,6.259,149.198
C09764=1143.515,10.975,-49.103,179.781,6.260,149.197
C09765=1143.510,11.225,-49.117,179.784,6.260,149.197
C09766=1143.505,11.475,-49.130,179.787,6.262,149.196
C09767=1143.500,11.724,-49.144,179.789,6.263,149.196
C09768=1143.495,11.974,-49.158,179.791,6.263,149.195
C09769=1143.489,12.224,-49.171,179.794,6.265,149.195
C09770=1143.485,12.473,-49.185,179.797,6.265,149.194
C09771=1143.479,12.722,-49.199,179.799,6.266,149.194
C09772=1143.474,12.972,-49.212,179.801,6.267,149.193
C09773=1143.469,13.222,-49.227,179.804,6.268,149.193
C09774=1143.464,13.471,-49.241,179.807,6.269,149.192
C09775=1143.459,13.721,-49.254,179.809,6.270,149.191
C09776=1143.454,13.971,-49.268,179.812,6.270,149.191
C09777=1143.449,14.220,-49.282,179.814,6.272,149.190
C09778=1143.444,14.469,-49.296,179.817,6.272,149.190
C09779=1143.438,14.720,-49.310,179.819,6.273,149.189
C09780=1143.434,14.968,-49.323,179.821,6.274,149.189
C09781=1143.429,15.218,-49.337,179.825,6.275,149.188
C09782=1143.423,15.467,-49.351,179.827,6.276,149.188
C09783=1143.418,15.718,-49.365,179.829,6.276,149.187
C09784=1143.413,15.967,-49.379,179.832,6.278,149.186
C09785=1143.408,16.217,-49.393,179.834,6.279,149.186
C09786=1143.403,16.466,-49.407,179.837,6.279,149.185
C09787=1143.398,16.715,-49.421,179.839,6.280,149.185
C09788=1143.393,16.966,-49.434,179.842,6.281,149.184
C09789=1143.387,17.215,-49.448,179.845,6.282,149.184
C09790=1143.382,17.464,-49.463,179.847,6.283,149.183
C09791=1143.377,17.714,-49.477,179.850,6.284,149.183
C09792=1143.372,17.963,-49.491,179.852,6.285,149.182
C09793=1143.367,18.213,-49.505,179.855,6.285,149.181
C09794=1143.363,18.462,-49.519,179.858,6.287,149.181
C09795=1143.357,18.711,-49.533,179.860,6.288,149.180
C09796=1143.352,18.962,-49.546,179.862,6.288,149.180
C09797=1143.347,19.211,-49.561,179.865,6.289,149.179
C09798=1143.342,19.461,-49.575,179.868,6.290,149.179
C09799=1143.336,19.710,-49.589,179.870,6.291,149.178
C09800=1143.331,19.960,-49.603,179.872,6.292,149.178
C09801=1143.327,20.209,-49.617,179.875,6.293,149.177
C09802=1143.322,20.459,-49.632,179.878,6.294,149.177
C09803=1143.316,20.708,-49.645,179.880,6.294,149.176
C09804=1143.311,20.958,-49.660,179.883,6.296,149.175
C09805=1143.306,21.208,-49.674,179.885,6.297,149.175
C09806=1143.301,21.457,-49.688,179.888,6.297,149.174
C09807=1143.296,21.706,-49.702,179.891,6.299,149.174
C09808=1143.291,21.956,-49.716,179.893,6.299,149.173
C09809=1143.286,22.206,-49.731,179.895,6.300,149.173
C09810=1143.281,22.455,-49.745,179.898,6.302,149.172
C09811=1143.276,22.705,-49.759,179.901,6.302,149.172
C09812=1143.270,22.954,-49.773,179.903,6.303,149.171
C09813=1143.265,23.204,-49.787,179.906,6.304,149.170
C09814=1143.260,23.454,-49.802,179.908,6.305,149.170
C09815=1143.255,23.703,-49.816,179.911,6.306,149.170
C09816=1143.250,23.953,-49.830,179.914,6.307,149.169
C09817=1143.245,24.202,-49.844,179.916,6.308,149.168
C09818=1143.240,24.452,-49.858,179.919,6.308,149.168
C09819=1143.235,24.701,-49.873,179.921,6.310,149.167
C09820=1143.230,24.951,-49.888,179.924,6.311,149.167
C09821=1143.225,25.200,-49.902,179.926,6.311,149.166
C09822=1143.220,25.449,-49.916,179.929,6.313,149.166
C09823=1143.215,25.699,-49.930,179.932,6.313,149.165
C09824=1143.209,25.949,-49.945,179.934,6.314,149.165
C09825=1143.204,26.199,-49.959,179.937,6.316,149.164
C09826=1143.200,26.448,-49.974,179.939,6.316,149.163
C09827=1143.195,26.697,-49.989,179.941,6.317,149.163
C09828=1143.189,26.946,-50.003,179.945,6.318,149.162
C09829=1143.184,27.215,-50.018,179.947,6.319,149.162
C09830=1143.178,27.485,-50.034,179.950,6.320,149.161
C09831=1143.173,27.754,-50.050,179.952,6.321,149.161
C09832=1143.167,28.023,-50.065,179.955,6.323,149.160
C09833=1143.162,28.272,-50.080,179.958,6.323,149.160
C09834=1143.158,28.522,-50.094,179.961,6.325,149.159
C09835=1143.152,28.772,-50.109,179.963,6.325,149.158
C09836=1143.147,29.021,-50.124,179.966,6.327,149.158
C09837=1143.142,29.270,-50.138,179.968,6.328,149.157
C09838=1143.137,29.520,-50.152,179.971,6.328,149.157
C09839=1143.132,29.769,-50.167,179.974,6.330,149.156
C09840=1143.127,30.019,-50.181,179.976,6.330,149.156
C09841=1143.121,30.269,-50.196,179.978,6.331,149.155
C09842=1143.117,30.518,-50.211,179.981,6.332,149.155
C09843=1143.112,30.767,-50.225,179.984,6.333,149.154
C09844=1143.107,31.017,-50.240,179.987,6.335,149.153
C09845=1143.101,31.267,-50.255,179.989,6.335,149.153
C09846=1143.096,31.516,-50.269,179.991,6.336,149.153
C09847=1143.092,31.766,-50.284,179.994,6.337,149.152
C09848=1143.087,32.015,-50.299,179.997,6.338,149.151
C09849=1143.081,32.265,-50.314,179.999,6.340,149.151
C09850=1143.076,32.515,-50.328,-179.998,6.340,149.150
C09851=1143.071,32.763,-50.342,-179.996,6.341,149.150
C09852=1143.066,33.013,-50.357,-179.993,6.342,149.149
C09853=1143.061,33.262,-50.372,-179.990,6.343,149.149
C09854=1143.056,33.512,-50.387,-179.988,6.345,149.148
C09855=1143.051,33.761,-50.402,-179.985,6.345,149.148
C09856=1143.045,34.011,-50.416,-179.983,6.346,149.147
C09857=1143.040,34.261,-50.431,-179.980,6.347,149.146
C09858=1143.036,34.510,-50.446,-179.977,6.348,149.146
C09859=1143.030,34.760,-50.461,-179.975,6.350,149.146
C09860=1143.025,35.009,-50.476,-179.972,6.350,149.145
C09861=1143.020,35.259,-50.490,-179.970,6.351,149.144
C09862=1143.015,35.508,-50.505,-179.967,6.353,149.144
C09863=1143.010,35.758,-50.520,-179.964,6.353,149.143
C09864=1143.005,36.007,-50.535,-179.962,6.355,149.143
C09865=1143.000,36.257,-50.550,-179.959,6.355,149.142
C09866=1142.995,36.506,-50.565,-179.956,6.357,149.142
C09867=1142.990,36.755,-50.580,-179.954,6.358,149.141
C09868=1142.985,37.005,-50.594,-179.951,6.358,149.141
C09869=1142.980,37.254,-50.609,-179.949,6.360,149.140
C09870=1142.974,37.504,-50.624,-179.947,6.361,149.140
C09871=1142.970,37.753,-50.639,-179.943,6.362,149.139
C09872=1142.965,38.003,-50.654,-179.941,6.363,149.139
C09873=1142.960,38.253,-50.670,-179.938,6.364,149.138
C09874=1142.955,38.502,-50.685,-179.936,6.365,149.137
C09875=1142.950,38.752,-50.699,-179.934,6.366,149.137
C09876=1142.945,39.001,-50.714,-179.930,6.367,149.136
C09877=1142.940,39.251,-50.730,-179.928,6.368,149.136
C09878=1142.935,39.501,-50.744,-179.925,6.370,149.135
C09879=1142.929,39.750,-50.760,-179.923,6.370,149.135
C09880=1142.925,39.999,-50.775,-179.920,6.372,149.134
C09881=1142.920,40.249,-50.789,-179.917,6.372,149.134
C09882=1142.914,40.498,-50.805,-179.915,6.374,149.133
C09883=1142.910,40.747,-50.820,-179.912,6.375,149.133
C09884=1142.904,40.997,-50.835,-179.910,6.375,149.132
C09885=1142.899,41.246,-50.850,-179.907,6.377,149.132
C09886=1142.895,41.496,-50.866,-179.905,6.378,149.131
C09887=1142.890,41.746,-50.881,-179.902,6.379,149.131
C09888=1142.884,41.996,-50.895,-179.899,6.380,149.130
C09889=1142.880,42.245,-50.910,-179.896,6.381,149.129
C09890=1142.874,42.494,-50.926,-179.894,6.382,149.129
C09891=1142.869,42.743,-50.942,-179.891,6.383,149.128
C09892=1142.864,42.993,-50.956,-179.889,6.384,149.128
C09893=1142.858,43.243,-50.971,-179.886,6.385,149.127
C09894=1142.854,43.492,-50.987,-179.884,6.386,149.127
C09895=1142.849,43.742,-51.002,-179.881,6.388,149.126
C09896=1142.844,43.991,-51.017,-179.878,6.388,149.126
C09897=1142.839,44.241,-51.032,-179.876,6.390,149.125
C09898=1142.834,44.490,-51.047,-179.873,6.390,149.125
C09899=1142.829,44.739,-51.063,-179.870,6.392,149.124
C09900=1142.824,44.989,-51.079,-179.868,6.393,149.124
C09901=1142.819,45.239,-51.094,-179.865,6.394,149.123
C09902=1142.814,45.488,-51.109,-179.863,6.395,149.123
C09903=1142.808,45.737,-51.125,-179.860,6.396,149.122
C09904=1142.804,45.986,-51.140,-179.857,6.397,149.122
C09905=1142.798,46.236,-51.155,-179.855,6.398,149.121
C09906=1142.794,46.486,-51.170,-179.852,6.399,149.120
C09907=1142.789,46.736,-51.186,-179.850,6.400,149.120
C09908=1142.783,46.985,-51.201,-179.847,6.402,149.120
C09909=1142.779,47.234,-51.216,-179.844,6.402,149.119
C09910=1142.774,47.484,-51.232,-179.842,6.404,149.118
C09911=1142.768,47.734,-51.248,-179.839,6.405,149.118
C09912=1142.764,47.983,-51.263,-179.836,6.406,149.117
C09913=1142.758,48.232,-51.278,-179.834,6.407,149.117
C09914=1142.753,48.482,-51.294,-179.831,6.408,149.116
C09915=1142.749,48.731,-51.309,-179.829,6.409,149.116
C09916=1142.744,48.981,-51.325,-179.826,6.411,149.115
C09917=1142.738,49.230,-51.341,-179.823,6.412,149.115
C09918=1142.734,49.479,-51.356,-179.820,6.413,149.114
C09919=1142.729,49.729,-51.372,-179.818,6.414,149.114
C09920=1142.723,49.979,-51.387,-179.815,6.415,149.113
C09921=1142.718,50.228,-51.403,-179.812,6.416,149.113
C09922=1142.714,50.477,-51.419,-179.810,6.417,149.112
C09923=1142.709,50.727,-51.434,-179.807,6.419,149.112
C09924=1142.703,50.976,-51.450,-179.805,6.419,149.111
C09925=1142.698,51.226,-51.466,-179.802,6.421,149.111
C09926=1142.694,51.475,-51.481,-179.799,6.421,149.110
C09927=1142.689,51.725,-51.497,-179.797,6.423,149.110
C09928=1142.683,51.974,-51.512,-179.794,6.424,149.109
C09929=1142.678,52.224,-51.528,-179.791,6.425,149.108
C09930=1142.673,52.474,-51.544,-179.789,6.426,149.108
C09931=1142.669,52.722,-51.559,-179.786,6.428,149.108
C09932=1142.663,52.972,-51.575,-179.784,6.428,149.107
C09933=1142.658,53.241,-51.592,-179.781,6.430,149.106
C09934=1142.653,53.509,-51.609,-179.778,6.431,149.106
C09935=1142.647,53.778,-51.626,-179.775,6.433,149.105
C09936=1142.641,54.047,-51.643,-179.772,6.433,149.105
C09937=1142.636,54.296,-51.659,-179.769,6.435,149.104
C09938=1142.632,54.545,-51.674,-179.767,6.437,149.104
C09939=1142.627,54.795,-51.690,-179.764,6.437,149.103
C09940=1142.622,55.044,-51.705,-179.761,6.439,149.103
C09941=1142.617,55.294,-51.722,-179.759,6.439,149.102
C09942=1142.612,55.543,-51.738,-179.756,6.441,149.102
C09943=1142.607,55.793,-51.754,-179.754,6.442,149.101
C09944=1142.602,56.042,-51.770,-179.751,6.443,149.101
C09945=1142.596,56.291,-51.786,-179.748,6.444,149.100
C09946=1142.592,56.541,-51.802,-179.746,6.445,149.100
C09947=1142.587,56.791,-51.817,-179.743,6.447,149.099
C09948=1142.582,57.039,-51.833,-179.740,6.447,149.098
C09949=1142.577,57.289,-51.849,-179.737,6.449,149.098
C09950=1142.572,57.539,-51.864,-179.735,6.450,149.098
C09951=1142.567,57.788,-51.881,-179.732,6.451,149.097
C09952=1142.562,58.038,-51.897,-179.730,6.452,149.096
C09953=1142.557,58.286,-51.913,-179.727,6.454,149.096
C09954=1142.552,58.537,-51.929,-179.724,6.455,149.095
C09955=1142.547,58.786,-51.944,-179.722,6.456,149.095
C09956=1142.542,59.035,-51.961,-179.719,6.458,149.095
C09957=1142.537,59.285,-51.977,-179.716,6.458,149.094
C09958=1142.532,59.534,-51.993,-179.714,6.460,149.093
C09959=1142.527,59.784,-52.009,-179.711,6.461,149.093
C09960=1142.522,60.033,-52.025,-179.708,6.462,149.092
C09961=1142.517,60.283,-52.041,-179.706,6.463,149.092
C09962=1142.512,60.532,-52.057,-179.703,6.464,149.091
C09963=1142.507,60.782,-52.074,-179.700,6.466,149.091
C09964=1142.502,61.031,-52.089,-179.698,6.466,149.090
C09965=1142.497,61.280,-52.106,-179.695,6.468,149.090
C09966=1142.492,61.530,-52.121,-179.692,6.469,149.089
C09967=1142.487,61.779,-52.138,-179.690,6.470,149.089
C09968=1142.482,62.028,-52.154,-179.687,6.472,149.088
C09969=1142.478,62.278,-52.170,-179.684,6.472,149.088
C09970=1142.472,62.527,-52.187,-179.682,6.474,149.087
C09971=1142.468,62.777,-52.203,-179.679,6.476,149.087
C09972=1142.462,63.026,-52.219,-179.677,6.476,149.086
C09973=1142.457,63.276,-52.235,-179.674,6.478,149.086
C09974=1142.452,63.525,-52.252,-179.671,6.479,149.085
C09975=1142.447,63.775,-52.268,-179.669,6.480,149.085
C09976=1142.442,64.024,-52.284,-179.665,6.481,149.084
C09977=1142.438,64.273,-52.301,-179.663,6.482,149.084
C09978=1142.432,64.523,-52.316,-179.661,6.484,149.083
C09979=1142.428,64.772,-52.333,-179.657,6.485,149.083
C09980=1142.423,65.021,-52.349,-179.655,6.486,149.082
C09981=1142.417,65.272,-52.366,-179.652,6.488,149.082
C09982=1142.412,65.520,-52.382,-179.649,6.489,149.081
C09983=1142.408,65.770,-52.399,-179.647,6.490,149.081
C09984=1142.402,66.019,-52.414,-179.644,6.492,149.080
C09985=1142.398,66.269,-52.431,-179.642,6.492,149.080
C09986=1142.393,66.517,-52.447,-179.639,6.494,149.079
C09987=1142.387,66.768,-52.464,-179.636,6.495,149.079
C09988=1142.383,67.017,-52.480,-179.634,6.496,149.078
C09989=1142.378,67.266,-52.497,-179.631,6.497,149.078
C09990=1142.373,67.516,-52.513,-179.628,6.499,149.077
C09991=1142.368,67.765,-52.529,-179.626,6.500,149.077
C09992=1142.362,68.015,-52.546,-179.623,6.501,149.076
C09993=1142.358,68.264,-52.563,-179.620,6.503,149.076
C09994=1142.353,68.513,-52.579,-179.618,6.504,149.075
C09995=1142.348,68.763,-52.596,-179.615,6.505,149.075
C09996=1142.342,69.012,-52.612,-179.612,6.507,149.074
//INST
///DATE 2021/06/15 17:27
///ATTR SC,RW,RJ
////FRAME ROBOT
///GROUP1 RB1
NOP
MOVL C00000 V=800.0 PL=0
MOVL C00001 V=800.0 PL=0
MOVL C00002 V=800.0 PL=0
MOVL C00003 V=800.0 PL=0
MOVL C00004 V=800.0 PL=0
MOVL C00005 V=800.0 PL=0
MOVL C00006 V=800.0 PL=0
MOVL C00007 V=800.0 PL=0
MOVL C00008 V=800.0 PL=0
MOVL C00009 V=800.0 PL=0
MOVL C00010 V=800.0 PL=0
MOVL C00011 V=800.0 PL=0
MOVL C00012 V=800.0 PL=0
MOVL C00013 V=800.0 PL=0
MOVL C00014 V=800.0 PL=0
MOVL C00015 V=800.0 PL=0
MOVL C00016 V=800.0 PL=0
MOVL C00017 V=800.0 PL=0
MOVL C00018 V=800.0 PL=0
MOVL C00019 V=800.0 PL=0
MOVL C00020 V=800.0 PL=0
MOVL C00021 V=800.0 PL=0
MOVL C00022 V=800.0 PL=0
MOVL C00023 V=800.0 PL=0
MOVL C00024 V=800.0 PL=0
MOVL C00025 V=800.0 PL=0
MOVL C00026 V=800.0 PL=0
MOVL C00027 V=800.0 PL=0
MOVL C00028 V=800.0 PL=0
MOVL C00029 V=800.0 PL=0
MOVL C00030 V=800.0 PL=0
MOVL C00031 V=800.0 PL=0
MOVL C00032 V=800.0 PL=0
MOVL C00033 V=800.0 PL=0
MOVL C00034 V=800.0 PL=0
MOVL C00035 V=800.0 PL=0
MOVL C00036 V=800.0 PL=0
MOVL C00037 V=800.0 PL=0
MOVL C00038 V=800.0 PL=0
MOVL C00039 V=800.0 PL=0
MOVL C00040 V=800.0 PL=0
MOVL C00041 V=800.0 PL=0
MOVL C00042 V=800.0 PL=0
MOVL C00043 V=800.0 PL=0
MOVL C00044 V=800.0 PL=0
MOVL C00045 V=800.0 PL=0
MOVL C00046 V=800.0 PL=0
MOVL C00047 V=800.0 PL=0
MOVL C00048 V=800.0 PL=0
MOVL C00049 V=800.0 PL=0
MOVL C00050 V=800.0 PL=0
MOVL C00051 V=800.0 PL=0
MOVL C00052 V=800.0 PL=0
MOVL C00053 V=800.0 PL=0
MOVL C00054 V=800.0 PL=0
MOVL C00055 V=800.0 PL=0
MOVL C00056 V=800.0 PL=0
MOVL C00057 V=800.0 PL=0
MOVL C00058 V=800.0 PL=0
MOVL C00059 V=800.0 PL=0
MOVL C00060 V=800.0 PL=0
MOVL C00061 V=800.0 PL=0
MOVL C00062 V=800.0 PL=0
MOVL C00063 V=800.0 PL=0
MOVL C00064 V=800.0 PL=0
MOVL C00065 V=800.0 PL=0
MOVL C00066 V=800.0 PL=0
MOVL C00067 V=800.0 PL=0
MOVL C00068 V=800.0 PL=0
MOVL C00069 V=800.0 PL=0
MOVL C00070 V=800.0 PL=0
MOVL C00071 V=800.0 PL=0
MOVL C00072 V=800.0 PL=0
MOVL C00073 V=800.0 PL=0
MOVL C00074 V=800.0 PL=0
MOVL C00075 V=800.0 PL=0
MOVL C00076 V=800.0 PL=0
MOVL C00077 V=800.0 PL=0
MOVL C00078 V=800.0 PL=0
MOVL C00079 V=800.0 PL=0
MOVL C00080 V=800.0 PL=0
MOVL C00081 V=800.0 PL=0
MOVL C00082 V=800.0 PL=0
MOVL C00083 V=800.0 PL=0
MOVL C00084 V=800.0 PL=0
MOVL C00085 V=800.0 PL=0
MOVL C00086 V=800.0 PL=0
MOVL C00087 V=800.0 PL=0
MOVL C00088 V=800.0 PL=0
MOVL C00089 V=800.0 PL=0
MOVL C00090 V=800.0 PL=0
MOVL C00091 V=800.0 PL=0
MOVL C00092 V=800.0 PL=0
MOVL C00093 V=800.0 PL=0
MOVL C00094 V=800.0 PL=0
MOVL C00095 V=800.0 PL=0
MOVL C00096 V=800.0 PL=0
MOVL C00097 V=800.0 PL=0
MOVL C00098 V=800.0 PL=0
MOVL C00099 V=800.0 PL=0
MOVL C00100 V=800.0 PL=0
MOVL C00101 V=800.0 PL=0
MOVL C00102 V=800.0 PL=0
MOVL C00103 V=800.0 PL=0
MOVL C00104 V=800.0 PL=0
MOVL C00105 V=800.0 PL=0
MOVL C00106 V=800.0 PL=0
MOVL C00107 V=800.0 PL=0
MOVL C00108 V=800.0 PL=0
MOVL C00109 V=800.0 PL=0
MOVL C00110 V=800.0 PL=0
MOVL C00111 V=800.0 PL=0
MOVL C00112 V=800.0 PL=0
MOVL C00113 V=800.0 PL=0
MOVL C00114 V=800.0 PL=0
MOVL C00115 V=800.0 PL=0
MOVL C00116 V=800.0 PL=0
MOVL C00117 V=800.0 PL=0
MOVL C00118 V=800.0 PL=0
MOVL C00119 V=800.0 PL=0
MOVL C00120 V=800.0 PL=0
MOVL C00121 V=800.0 PL=0
MOVL C00122 V=800.0 PL=0
MOVL C00123 V=800.0 PL=0
MOVL C00124 V=800.0 PL=0
MOVL C00125 V=800.0 PL=0
MOVL C00126 V=800.0 PL=0
MOVL C00127 V=800.0 PL=0
MOVL C00128 V=800.0 PL=0
MOVL C00129 V=800.0 PL=0
MOVL C00130 V=800.0 PL=0
MOVL C00131 V=800.0 PL=0
MOVL C00132 V=800.0 PL=0
MOVL C00133 V=800.0 PL=0
MOVL C00134 V=800.0 PL=0
MOVL C00135 V=800.0 PL=0
MOVL C00136 V=800.0 PL=0
MOVL C00137 V=800.0 PL=0
MOVL C00138 V=800.0 PL=0
MOVL C00139 V=800.0 PL=0
MOVL C00140 V=800.0 PL=0
MOVL C00141 V=800.0 PL=0
MOVL C00142 V=800.0 PL=0
MOVL C00143 V=800.0 PL=0
MOVL C00144 V=800.0 PL=0
MOVL C00145 V=800.0 PL=0
MOVL C00146 V=800.0 PL=0
MOVL C00147 V=800.0 PL=0
MOVL C00148 V=800.0 PL=0
MOVL C00149 V=800.0 PL=0
MOVL C00150 V=800.0 PL=0
MOVL C00151 V=800.0 PL=0
MOVL C00152 V=800.0 PL=0
MOVL C00153 V=800.0 PL=0
MOVL C00154 V=800.0 PL=0
MOVL C00155 V=800.0 PL=0
MOVL C00156 V=800.0 PL=0
MOVL C00157 V=800.0 PL=0
MOVL C00158 V=800.0 PL=0
MOVL C00159 V=800.0 PL=0
MOVL C00160 V=800.0 PL=0
MOVL C00161 V=800.0 PL=0
MOVL C00162 V=800.0 PL=0
MOVL C00163 V=800.0 PL=0
MOVL C00164 V=800.0 PL=0
MOVL C00165 V=800.0 PL=0
MOVL C00166 V=800.0 PL=0
MOVL C00167 V=800.0 PL=0
MOVL C00168 V=800.0 PL=0
MOVL C00169 V=800.0 PL=0
MOVL C00170 V=800.0 PL=0
MOVL C00171 V=800.0 PL=0
MOVL C00172 V=800.0 PL=0
MOVL C00173 V=800.0 PL=0
MOVL C00174 V=800.0 PL=0
MOVL C00175 V=800.0 PL=0
MOVL C00176 V=800.0 PL=0
MOVL C00177 V=800.0 PL=0
MOVL C00178 V=800.0 PL=0
MOVL C00179 V=800.0 PL=0
MOVL C00180 V=800.0 PL=0
MOVL C00181 V=800.0 PL=0
MOVL C00182 V=800.0 PL=0
MOVL C00183 V=800.0 PL=0
MOVL C00184 V=800.0 PL=0
MOVL C00185 V=800.0 PL=0
MOVL C00186 V=800.0 PL=0
MOVL C00187 V=800.0 PL=0
MOVL C00188 V=800.0 PL=0
MOVL C00189 V=800.0 PL=0
MOVL C00190 V=800.0 PL=0
MOVL C00191 V=800.0 PL=0
MOVL C00192 V=800.0 PL=0
MOVL C00193 V=800.0 PL=0
MOVL C00194 V=800.0 PL=0
MOVL C00195 V=800.0 PL=0
MOVL C00196 V=800.0 PL=0
MOVL C00197 V=800.0 PL=0
MOVL C00198 V=800.0 PL=0
MOVL C00199 V=800.0 PL=0
MOVL C00200 V=800.0 PL=0
MOVL C00201 V=800.0 PL=0
MOVL C00202 V=800.0 PL=0
MOVL C00203 V=800.0 PL=0
MOVL C00204 V=800.0 PL=0
MOVL C00205 V=800.0 PL=0
MOVL C00206 V=800.0 PL=0
MOVL C00207 V=800.0 PL=0
MOVL C00208 V=800.0 PL=0
MOVL C00209 V=800.0 PL=0
MOVL C00210 V=800.0 PL=0
MOVL C00211 V=800.0 PL=0
MOVL C00212 V=800.0 PL=0
MOVL C00213 V=800.0 PL=0
MOVL C00214 V=800.0 PL=0
MOVL C00215 V=800.0 PL=0
MOVL C00216 V=800.0 PL=0
MOVL C00217 V=800.0 PL=0
MOVL C00218 V=800.0 PL=0
MOVL C00219 V=800.0 PL=0
MOVL C00220 V=800.0 PL=0
MOVL C00221 V=800.0 PL=0
MOVL C00222 V=800.0 PL=0
MOVL C00223 V=800.0 PL=0
MOVL C00224 V=800.0 PL=0
MOVL C00225 V=800.0 PL=0
MOVL C00226 V=800.0 PL=0
MOVL C00227 V=800.0 PL=0
MOVL C00228 V=800.0 PL=0
MOVL C00229 V=800.0 PL=0
MOVL C00230 V=800.0 PL=0
MOVL C00231 V=800.0 PL=0
MOVL C00232 V=800.0 PL=0
MOVL C00233 V=800.0 PL=0
MOVL C00234 V=800.0 PL=0
MOVL C00235 V=800.0 PL=0
MOVL C00236 V=800.0 PL=0
MOVL C00237 V=800.0 PL=0
MOVL C00238 V=800.0 PL=0
MOVL C00239 V=800.0 PL=0
MOVL C00240 V=800.0 PL=0
MOVL C00241 V=800.0 PL=0
MOVL C00242 V=800.0 PL=0
MOVL C00243 V=800.0 PL=0
MOVL C00244 V=800.0 PL=0
MOVL C00245 V=800.0 PL=0
MOVL C00246 V=800.0 PL=0
MOVL C00247 V=800.0 PL=0
MOVL C00248 V=800.0 PL=0
MOVL C00249 V=800.0 PL=0
MOVL C00250 V=800.0 PL=0
MOVL C00251 V=800.0 PL=0
MOVL C00252 V=800.0 PL=0
MOVL C00253 V=800.0 PL=0
MOVL C00254 V=800.0 PL=0
MOVL C00255 V=800.0 PL=0
MOVL C00256 V=800.0 PL=0
MOVL C00257 V=800.0 PL=0
MOVL C00258 V=800.0 PL=0
MOVL C00259 V=800.0 PL=0
MOVL C00260 V=800.0 PL=0
MOVL C00261 V=800.0 PL=0
MOVL C00262 V=800.0 PL=0
MOVL C00263 V=800.0 PL=0
MOVL C00264 V=800.0 PL=0
MOVL C00265 V=800.0 PL=0
MOVL C00266 V=800.0 PL=0
MOVL C00267 V=800.0 PL=0
MOVL C00268 V=800.0 PL=0
MOVL C00269 V=800.0 PL=0
MOVL C00270 V=800.0 PL=0
MOVL C00271 V=800.0 PL=0
MOVL C00272 V=800.0 PL=0
MOVL C00273 V=800.0 PL=0
MOVL C00274 V=800.0 PL=0
MOVL C00275 V=800.0 PL=0
MOVL C00276 V=800.0 PL=0
MOVL C00277 V=800.0 PL=0
MOVL C00278 V=800.0 PL=0
MOVL C00279 V=800.0 PL=0
MOVL C00280 V=800.0 PL=0
MOVL C00281 V=800.0 PL=0
MOVL C00282 V=800.0 PL=0
MOVL C00283 V=800.0 PL=0
MOVL C00284 V=800.0 PL=0
MOVL C00285 V=800.0 PL=0
MOVL C00286 V=800.0 PL=0
MOVL C00287 V=800.0 PL=0
MOVL C00288 V=800.0 PL=0
MOVL C00289 V=800.0 PL=0
MOVL C00290 V=800.0 PL=0
MOVL C00291 V=800.0 PL=0
MOVL C00292 V=800.0 PL=0
MOVL C00293 V=800.0 PL=0
MOVL C00294 V=800.0 PL=0
MOVL C00295 V=800.0 PL=0
MOVL C00296 V=800.0 PL=0
MOVL C00297 V=800.0 PL=0
MOVL C00298 V=800.0 PL=0
MOVL C00299 V=800.0 PL=0
MOVL C00300 V=800.0 PL=0
MOVL C00301 V=800.0 PL=0
MOVL C00302 V=800.0 PL=0
MOVL C00303 V=800.0 PL=0
MOVL C00304 V=800.0 PL=0
MOVL C00305 V=800.0 PL=0
MOVL C00306 V=800.0 PL=0
MOVL C00307 V=800.0 PL=0
MOVL C00308 V=800.0 PL=0
MOVL C00309 V=800.0 PL=0
MOVL C00310 V=800.0 PL=0
MOVL C00311 V=800.0 PL=0
MOVL C00312 V=800.0 PL=0
MOVL C00313 V=800.0 PL=0
MOVL C00314 V=800.0 PL=0
MOVL C00315 V=800.0 PL=0
MOVL C00316 V=800.0 PL=0
MOVL C00317 V=800.0 PL=0
MOVL C00318 V=800.0 PL=0
MOVL C00319 V=800.0 PL=0
MOVL C00320 V=800.0 PL=0
MOVL C00321 V=800.0 PL=0
MOVL C00322 V=800.0 PL=0
MOVL C00323 V=800.0 PL=0
MOVL C00324 V=800.0 PL=0
MOVL C00325 V=800.0 PL=0
MOVL C00326 V=800.0 PL=0
MOVL C00327 V=800.0 PL=0
MOVL C00328 V=800.0 PL=0
MOVL C00329 V=800.0 PL=0
MOVL C00330 V=800.0 PL=0
MOVL C00331 V=800.0 PL=0
MOVL C00332 V=800.0 PL=0
MOVL C00333 V=800.0 PL=0
MOVL C00334 V=800.0 PL=0
MOVL C00335 V=800.0 PL=0
MOVL C00336 V=800.0 PL=0
MOVL C00337 V=800.0 PL=0
MOVL C00338 V=800.0 PL=0
MOVL C00339 V=800.0 PL=0
MOVL C00340 V=800.0 PL=0
MOVL C00341 V=800.0 PL=0
MOVL C00342 V=800.0 PL=0
MOVL C00343 V=800.0 PL=0
MOVL C00344 V=800.0 PL=0
MOVL C00345 V=800.0 PL=0
MOVL C00346 V=800.0 PL=0
MOVL C00347 V=800.0 PL=0
MOVL C00348 V=800.0 PL=0
MOVL C00349 V=800.0 PL=0
MOVL C00350 V=800.0 PL=0
MOVL C00351 V=800.0 PL=0
MOVL C00352 V=800.0 PL=0
MOVL C00353 V=800.0 PL=0
MOVL C00354 V=800.0 PL=0
MOVL C00355 V=800.0 PL=0
MOVL C00356 V=800.0 PL=0
MOVL C00357 V=800.0 PL=0
MOVL C00358 V=800.0 PL=0
MOVL C00359 V=800.0 PL=0
MOVL C00360 V=800.0 PL=0
MOVL C00361 V=800.0 PL=0
MOVL C00362 V=800.0 PL=0
MOVL C00363 V=800.0 PL=0
MOVL C00364 V=800.0 PL=0
MOVL C00365 V=800.0 PL=0
MOVL C00366 V=800.0 PL=0
MOVL C00367 V=800.0 PL=0
MOVL C00368 V=800.0 PL=0
MOVL C00369 V=800.0 PL=0
MOVL C00370 V=800.0 PL=0
MOVL C00371 V=800.0 PL=0
MOVL C00372 V=800.0 PL=0
MOVL C00373 V=800.0 PL=0
MOVL C00374 V=800.0 PL=0
MOVL C00375 V=800.0 PL=0
MOVL C00376 V=800.0 PL=0
MOVL C00377 V=800.0 PL=0
MOVL C00378 V=800.0 PL=0
MOVL C00379 V=800.0 PL=0
MOVL C00380 V=800.0 PL=0
MOVL C00381 V=800.0 PL=0
MOVL C00382 V=800.0 PL=0
MOVL C00383 V=800.0 PL=0
MOVL C00384 V=800.0 PL=0
MOVL C00385 V=800.0 PL=0
MOVL C00386 V=800.0 PL=0
MOVL C00387 V=800.0 PL=0
MOVL C00388 V=800.0 PL=0
MOVL C00389 V=800.0 PL=0
MOVL C00390 V=800.0 PL=0
MOVL C00391 V=800.0 PL=0
MOVL C00392 V=800.0 PL=0
MOVL C00393 V=800.0 PL=0
MOVL C00394 V=800.0 PL=0
MOVL C00395 V=800.0 PL=0
MOVL C00396 V=800.0 PL=0
MOVL C00397 V=800.0 PL=0
MOVL C00398 V=800.0 PL=0
MOVL C00399 V=800.0 PL=0
MOVL C00400 V=800.0 PL=0
MOVL C00401 V=800.0 PL=0
MOVL C00402 V=800.0 PL=0
MOVL C00403 V=800.0 PL=0
MOVL C00404 V=800.0 PL=0
MOVL C00405 V=800.0 PL=0
MOVL C00406 V=800.0 PL=0
MOVL C00407 V=800.0 PL=0
MOVL C00408 V=800.0 PL=0
MOVL C00409 V=800.0 PL=0
MOVL C00410 V=800.0 PL=0
MOVL C00411 V=800.0 PL=0
MOVL C00412 V=800.0 PL=0
MOVL C00413 V=800.0 PL=0
MOVL C00414 V=800.0 PL=0
MOVL C00415 V=800.0 PL=0
MOVL C00416 V=800.0 PL=0
MOVL C00417 V=800.0 PL=0
MOVL C00418 V=800.0 PL=0
MOVL C00419 V=800.0 PL=0
MOVL C00420 V=800.0 PL=0
MOVL C00421 V=800.0 PL=0
MOVL C00422 V=800.0 PL=0
MOVL C00423 V=800.0 PL=0
MOVL C00424 V=800.0 PL=0
MOVL C00425 V=800.0 PL=0
MOVL C00426 V=800.0 PL=0
MOVL C00427 V=800.0 PL=0
MOVL C00428 V=800.0 PL=0
MOVL C00429 V=800.0 PL=0
MOVL C00430 V=800.0 PL=0
MOVL C00431 V=800.0 PL=0
MOVL C00432 V=800.0 PL=0
MOVL C00433 V=800.0 PL=0
MOVL C00434 V=800.0 PL=0
MOVL C00435 V=800.0 PL=0
MOVL C00436 V=800.0 PL=0
MOVL C00437 V=800.0 PL=0
MOVL C00438 V=800.0 PL=0
MOVL C00439 V=800.0 PL=0
MOVL C00440 V=800.0 PL=0
MOVL C00441 V=800.0 PL=0
MOVL C00442 V=800.0 PL=0
MOVL C00443 V=800.0 PL=0
MOVL C00444 V=800.0 PL=0
MOVL C00445 V=800.0 PL=0
MOVL C00446 V=800.0 PL=0
MOVL C00447 V=800.0 PL=0
MOVL C00448 V=800.0 PL=0
MOVL C00449 V=800.0 PL=0
MOVL C00450 V=800.0 PL=0
MOVL C00451 V=800.0 PL=0
MOVL C00452 V=800.0 PL=0
MOVL C00453 V=800.0 PL=0
MOVL C00454 V=800.0 PL=0
MOVL C00455 V=800.0 PL=0
MOVL C00456 V=800.0 PL=0
MOVL C00457 V=800.0 PL=0
MOVL C00458 V=800.0 PL=0
MOVL C00459 V=800.0 PL=0
MOVL C00460 V=800.0 PL=0
MOVL C00461 V=800.0 PL=0
MOVL C00462 V=800.0 PL=0
MOVL C00463 V=800.0 PL=0
MOVL C00464 V=800.0 PL=0
MOVL C00465 V=800.0 PL=0
MOVL C00466 V=800.0 PL=0
MOVL C00467 V=800.0 PL=0
MOVL C00468 V=800.0 PL=0
MOVL C00469 V=800.0 PL=0
MOVL C00470 V=800.0 PL=0
MOVL C00471 V=800.0 PL=0
MOVL C00472 V=800.0 PL=0
MOVL C00473 V=800.0 PL=0
MOVL C00474 V=800.0 PL=0
MOVL C00475 V=800.0 PL=0
MOVL C00476 V=800.0 PL=0
MOVL C00477 V=800.0 PL=0
MOVL C00478 V=800.0 PL=0
MOVL C00479 V=800.0 PL=0
MOVL C00480 V=800.0 PL=0
MOVL C00481 V=800.0 PL=0
MOVL C00482 V=800.0 PL=0
MOVL C00483 V=800.0 PL=0
MOVL C00484 V=800.0 PL=0
MOVL C00485 V=800.0 PL=0
MOVL C00486 V=800.0 PL=0
MOVL C00487 V=800.0 PL=0
MOVL C00488 V=800.0 PL=0
MOVL C00489 V=800.0 PL=0
MOVL C00490 V=800.0 PL=0
MOVL C00491 V=800.0 PL=0
MOVL C00492 V=800.0 PL=0
MOVL C00493 V=800.0 PL=0
MOVL C00494 V=800.0 PL=0
MOVL C00495 V=800.0 PL=0
MOVL C00496 V=800.0 PL=0
MOVL C00497 V=800.0 PL=0
MOVL C00498 V=800.0 PL=0
MOVL C00499 V=800.0 PL=0
MOVL C00500 V=800.0 PL=0
MOVL C00501 V=800.0 PL=0
MOVL C00502 V=800.0 PL=0
MOVL C00503 V=800.0 PL=0
MOVL C00504 V=800.0 PL=0
MOVL C00505 V=800.0 PL=0
MOVL C00506 V=800.0 PL=0
MOVL C00507 V=800.0 PL=0
MOVL C00508 V=800.0 PL=0
MOVL C00509 V=800.0 PL=0
MOVL C00510 V=800.0 PL=0
MOVL C00511 V=800.0 PL=0
MOVL C00512 V=800.0 PL=0
MOVL C00513 V=800.0 PL=0
MOVL C00514 V=800.0 PL=0
MOVL C00515 V=800.0 PL=0
MOVL C00516 V=800.0 PL=0
MOVL C00517 V=800.0 PL=0
MOVL C00518 V=800.0 PL=0
MOVL C00519 V=800.0 PL=0
MOVL C00520 V=800.0 PL=0
MOVL C00521 V=800.0 PL=0
MOVL C00522 V=800.0 PL=0
MOVL C00523 V=800.0 PL=0
MOVL C00524 V=800.0 PL=0
MOVL C00525 V=800.0 PL=0
MOVL C00526 V=800.0 PL=0
MOVL C00527 V=800.0 PL=0
MOVL C00528 V=800.0 PL=0
MOVL C00529 V=800.0 PL=0
MOVL C00530 V=800.0 PL=0
MOVL C00531 V=800.0 PL=0
MOVL C00532 V=800.0 PL=0
MOVL C00533 V=800.0 PL=0
MOVL C00534 V=800.0 PL=0
MOVL C00535 V=800.0 PL=0
MOVL C00536 V=800.0 PL=0
MOVL C00537 V=800.0 PL=0
MOVL C00538 V=800.0 PL=0
MOVL C00539 V=800.0 PL=0
MOVL C00540 V=800.0 PL=0
MOVL C00541 V=800.0 PL=0
MOVL C00542 V=800.0 PL=0
MOVL C00543 V=800.0 PL=0
MOVL C00544 V=800.0 PL=0
MOVL C00545 V=800.0 PL=0
MOVL C00546 V=800.0 PL=0
MOVL C00547 V=800.0 PL=0
MOVL C00548 V=800.0 PL=0
MOVL C00549 V=800.0 PL=0
MOVL C00550 V=800.0 PL=0
MOVL C00551 V=800.0 PL=0
MOVL C00552 V=800.0 PL=0
MOVL C00553 V=800.0 PL=0
MOVL C00554 V=800.0 PL=0
MOVL C00555 V=800.0 PL=0
MOVL C00556 V=800.0 PL=0
MOVL C00557 V=800.0 PL=0
MOVL C00558 V=800.0 PL=0
MOVL C00559 V=800.0 PL=0
MOVL C00560 V=800.0 PL=0
MOVL C00561 V=800.0 PL=0
MOVL C00562 V=800.0 PL=0
MOVL C00563 V=800.0 PL=0
MOVL C00564 V=800.0 PL=0
MOVL C00565 V=800.0 PL=0
MOVL C00566 V=800.0 PL=0
MOVL C00567 V=800.0 PL=0
MOVL C00568 V=800.0 PL=0
MOVL C00569 V=800.0 PL=0
MOVL C00570 V=800.0 PL=0
MOVL C00571 V=800.0 PL=0
MOVL C00572 V=800.0 PL=0
MOVL C00573 V=800.0 PL=0
MOVL C00574 V=800.0 PL=0
MOVL C00575 V=800.0 PL=0
MOVL C00576 V=800.0 PL=0
MOVL C00577 V=800.0 PL=0
MOVL C00578 V=800.0 PL=0
MOVL C00579 V=800.0 PL=0
MOVL C00580 V=800.0 PL=0
MOVL C00581 V=800.0 PL=0
MOVL C00582 V=800.0 PL=0
MOVL C00583 V=800.0 PL=0
MOVL C00584 V=800.0 PL=0
MOVL C00585 V=800.0 PL=0
MOVL C00586 V=800.0 PL=0
MOVL C00587 V=800.0 PL=0
MOVL C00588 V=800.0 PL=0
MOVL C00589 V=800.0 PL=0
MOVL C00590 V=800.0 PL=0
MOVL C00591 V=800.0 PL=0
MOVL C00592 V=800.0 PL=0
MOVL C00593 V=800.0 PL=0
MOVL C00594 V=800.0 PL=0
MOVL C00595 V=800.0 PL=0
MOVL C00596 V=800.0 PL=0
MOVL C00597 V=800.0 PL=0
MOVL C00598 V=800.0 PL=0
MOVL C00599 V=800.0 PL=0
MOVL C00600 V=800.0 PL=0
MOVL C00601 V=800.0 PL=0
MOVL C00602 V=800.0 PL=0
MOVL C00603 V=800.0 PL=0
MOVL C00604 V=800.0 PL=0
MOVL C00605 V=800.0 PL=0
MOVL C00606 V=800.0 PL=0
MOVL C00607 V=800.0 PL=0
MOVL C00608 V=800.0 PL=0
MOVL C00609 V=800.0 PL=0
MOVL C00610 V=800.0 PL=0
MOVL C00611 V=800.0 PL=0
MOVL C00612 V=800.0 PL=0
MOVL C00613 V=800.0 PL=0
MOVL C00614 V=800.0 PL=0
MOVL C00615 V=800.0 PL=0
MOVL C00616 V=800.0 PL=0
MOVL C00617 V=800.0 PL=0
MOVL C00618 V=800.0 PL=0
MOVL C00619 V=800.0 PL=0
MOVL C00620 V=800.0 PL=0
MOVL C00621 V=800.0 PL=0
MOVL C00622 V=800.0 PL=0
MOVL C00623 V=800.0 PL=0
MOVL C00624 V=800.0 PL=0
MOVL C00625 V=800.0 PL=0
MOVL C00626 V=800.0 PL=0
MOVL C00627 V=800.0 PL=0
MOVL C00628 V=800.0 PL=0
MOVL C00629 V=800.0 PL=0
MOVL C00630 V=800.0 PL=0
MOVL C00631 V=800.0 PL=0
MOVL C00632 V=800.0 PL=0
MOVL C00633 V=800.0 PL=0
MOVL C00634 V=800.0 PL=0
MOVL C00635 V=800.0 PL=0
MOVL C00636 V=800.0 PL=0
MOVL C00637 V=800.0 PL=0
MOVL C00638 V=800.0 PL=0
MOVL C00639 V=800.0 PL=0
MOVL C00640 V=800.0 PL=0
MOVL C00641 V=800.0 PL=0
MOVL C00642 V=800.0 PL=0
MOVL C00643 V=800.0 PL=0
MOVL C00644 V=800.0 PL=0
MOVL C00645 V=800.0 PL=0
MOVL C00646 V=800.0 PL=0
MOVL C00647 V=800.0 PL=0
MOVL C00648 V=800.0 PL=0
MOVL C00649 V=800.0 PL=0
MOVL C00650 V=800.0 PL=0
MOVL C00651 V=800.0 PL=0
MOVL C00652 V=800.0 PL=0
MOVL C00653 V=800.0 PL=0
MOVL C00654 V=800.0 PL=0
MOVL C00655 V=800.0 PL=0
MOVL C00656 V=800.0 PL=0
MOVL C00657 V=800.0 PL=0
MOVL C00658 V=800.0 PL=0
MOVL C00659 V=800.0 PL=0
MOVL C00660 V=800.0 PL=0
MOVL C00661 V=800.0 PL=0
MOVL C00662 V=800.0 PL=0
MOVL C00663 V=800.0 PL=0
MOVL C00664 V=800.0 PL=0
MOVL C00665 V=800.0 PL=0
MOVL C00666 V=800.0 PL=0
MOVL C00667 V=800.0 PL=0
MOVL C00668 V=800.0 PL=0
MOVL C00669 V=800.0 PL=0
MOVL C00670 V=800.0 PL=0
MOVL C00671 V=800.0 PL=0
MOVL C00672 V=800.0 PL=0
MOVL C00673 V=800.0 PL=0
MOVL C00674 V=800.0 PL=0
MOVL C00675 V=800.0 PL=0
MOVL C00676 V=800.0 PL=0
MOVL C00677 V=800.0 PL=0
MOVL C00678 V=800.0 PL=0
MOVL C00679 V=800.0 PL=0
MOVL C00680 V=800.0 PL=0
MOVL C00681 V=800.0 PL=0
MOVL C00682 V=800.0 PL=0
MOVL C00683 V=800.0 PL=0
MOVL C00684 V=800.0 PL=0
MOVL C00685 V=800.0 PL=0
MOVL C00686 V=800.0 PL=0
MOVL C00687 V=800.0 PL=0
MOVL C00688 V=800.0 PL=0
MOVL C00689 V=800.0 PL=0
MOVL C00690 V=800.0 PL=0
MOVL C00691 V=800.0 PL=0
MOVL C00692 V=800.0 PL=0
MOVL C00693 V=800.0 PL=0
MOVL C00694 V=800.0 PL=0
MOVL C00695 V=800.0 PL=0
MOVL C00696 V=800.0 PL=0
MOVL C00697 V=800.0 PL=0
MOVL C00698 V=800.0 PL=0
MOVL C00699 V=800.0 PL=0
MOVL C00700 V=800.0 PL=0
MOVL C00701 V=800.0 PL=0
MOVL C00702 V=800.0 PL=0
MOVL C00703 V=800.0 PL=0
MOVL C00704 V=800.0 PL=0
MOVL C00705 V=800.0 PL=0
MOVL C00706 V=800.0 PL=0
MOVL C00707 V=800.0 PL=0
MOVL C00708 V=800.0 PL=0
MOVL C00709 V=800.0 PL=0
MOVL C00710 V=800.0 PL=0
MOVL C00711 V=800.0 PL=0
MOVL C00712 V=800.0 PL=0
MOVL C00713 V=800.0 PL=0
MOVL C00714 V=800.0 PL=0
MOVL C00715 V=800.0 PL=0
MOVL C00716 V=800.0 PL=0
MOVL C00717 V=800.0 PL=0
MOVL C00718 V=800.0 PL=0
MOVL C00719 V=800.0 PL=0
MOVL C00720 V=800.0 PL=0
MOVL C00721 V=800.0 PL=0
MOVL C00722 V=800.0 PL=0
MOVL C00723 V=800.0 PL=0
MOVL C00724 V=800.0 PL=0
MOVL C00725 V=800.0 PL=0
MOVL C00726 V=800.0 PL=0
MOVL C00727 V=800.0 PL=0
MOVL C00728 V=800.0 PL=0
MOVL C00729 V=800.0 PL=0
MOVL C00730 V=800.0 PL=0
MOVL C00731 V=800.0 PL=0
MOVL C00732 V=800.0 PL=0
MOVL C00733 V=800.0 PL=0
MOVL C00734 V=800.0 PL=0
MOVL C00735 V=800.0 PL=0
MOVL C00736 V=800.0 PL=0
MOVL C00737 V=800.0 PL=0
MOVL C00738 V=800.0 PL=0
MOVL C00739 V=800.0 PL=0
MOVL C00740 V=800.0 PL=0
MOVL C00741 V=800.0 PL=0
MOVL C00742 V=800.0 PL=0
MOVL C00743 V=800.0 PL=0
MOVL C00744 V=800.0 PL=0
MOVL C00745 V=800.0 PL=0
MOVL C00746 V=800.0 PL=0
MOVL C00747 V=800.0 PL=0
MOVL C00748 V=800.0 PL=0
MOVL C00749 V=800.0 PL=0
MOVL C00750 V=800.0 PL=0
MOVL C00751 V=800.0 PL=0
MOVL C00752 V=800.0 PL=0
MOVL C00753 V=800.0 PL=0
MOVL C00754 V=800.0 PL=0
MOVL C00755 V=800.0 PL=0
MOVL C00756 V=800.0 PL=0
MOVL C00757 V=800.0 PL=0
MOVL C00758 V=800.0 PL=0
MOVL C00759 V=800.0 PL=0
MOVL C00760 V=800.0 PL=0
MOVL C00761 V=800.0 PL=0
MOVL C00762 V=800.0 PL=0
MOVL C00763 V=800.0 PL=0
MOVL C00764 V=800.0 PL=0
MOVL C00765 V=800.0 PL=0
MOVL C00766 V=800.0 PL=0
MOVL C00767 V=800.0 PL=0
MOVL C00768 V=800.0 PL=0
MOVL C00769 V=800.0 PL=0
MOVL C00770 V=800.0 PL=0
MOVL C00771 V=800.0 PL=0
MOVL C00772 V=800.0 PL=0
MOVL C00773 V=800.0 PL=0
MOVL C00774 V=800.0 PL=0
MOVL C00775 V=800.0 PL=0
MOVL C00776 V=800.0 PL=0
MOVL C00777 V=800.0 PL=0
MOVL C00778 V=800.0 PL=0
MOVL C00779 V=800.0 PL=0
MOVL C00780 V=800.0 PL=0
MOVL C00781 V=800.0 PL=0
MOVL C00782 V=800.0 PL=0
MOVL C00783 V=800.0 PL=0
MOVL C00784 V=800.0 PL=0
MOVL C00785 V=800.0 PL=0
MOVL C00786 V=800.0 PL=0
MOVL C00787 V=800.0 PL=0
MOVL C00788 V=800.0 PL=0
MOVL C00789 V=800.0 PL=0
MOVL C00790 V=800.0 PL=0
MOVL C00791 V=800.0 PL=0
MOVL C00792 V=800.0 PL=0
MOVL C00793 V=800.0 PL=0
MOVL C00794 V=800.0 PL=0
MOVL C00795 V=800.0 PL=0
MOVL C00796 V=800.0 PL=0
MOVL C00797 V=800.0 PL=0
MOVL C00798 V=800.0 PL=0
MOVL C00799 V=800.0 PL=0
MOVL C00800 V=800.0 PL=0
MOVL C00801 V=800.0 PL=0
MOVL C00802 V=800.0 PL=0
MOVL C00803 V=800.0 PL=0
MOVL C00804 V=800.0 PL=0
MOVL C00805 V=800.0 PL=0
MOVL C00806 V=800.0 PL=0
MOVL C00807 V=800.0 PL=0
MOVL C00808 V=800.0 PL=0
MOVL C00809 V=800.0 PL=0
MOVL C00810 V=800.0 PL=0
MOVL C00811 V=800.0 PL=0
MOVL C00812 V=800.0 PL=0
MOVL C00813 V=800.0 PL=0
MOVL C00814 V=800.0 PL=0
MOVL C00815 V=800.0 PL=0
MOVL C00816 V=800.0 PL=0
MOVL C00817 V=800.0 PL=0
MOVL C00818 V=800.0 PL=0
MOVL C00819 V=800.0 PL=0
MOVL C00820 V=800.0 PL=0
MOVL C00821 V=800.0 PL=0
MOVL C00822 V=800.0 PL=0
MOVL C00823 V=800.0 PL=0
MOVL C00824 V=800.0 PL=0
MOVL C00825 V=800.0 PL=0
MOVL C00826 V=800.0 PL=0
MOVL C00827 V=800.0 PL=0
MOVL C00828 V=800.0 PL=0
MOVL C00829 V=800.0 PL=0
MOVL C00830 V=800.0 PL=0
MOVL C00831 V=800.0 PL=0
MOVL C00832 V=800.0 PL=0
MOVL C00833 V=800.0 PL=0
MOVL C00834 V=800.0 PL=0
MOVL C00835 V=800.0 PL=0
MOVL C00836 V=800.0 PL=0
MOVL C00837 V=800.0 PL=0
MOVL C00838 V=800.0 PL=0
MOVL C00839 V=800.0 PL=0
MOVL C00840 V=800.0 PL=0
MOVL C00841 V=800.0 PL=0
MOVL C00842 V=800.0 PL=0
MOVL C00843 V=800.0 PL=0
MOVL C00844 V=800.0 PL=0
MOVL C00845 V=800.0 PL=0
MOVL C00846 V=800.0 PL=0
MOVL C00847 V=800.0 PL=0
MOVL C00848 V=800.0 PL=0
MOVL C00849 V=800.0 PL=0
MOVL C00850 V=800.0 PL=0
MOVL C00851 V=800.0 PL=0
MOVL C00852 V=800.0 PL=0
MOVL C00853 V=800.0 PL=0
MOVL C00854 V=800.0 PL=0
MOVL C00855 V=800.0 PL=0
MOVL C00856 V=800.0 PL=0
MOVL C00857 V=800.0 PL=0
MOVL C00858 V=800.0 PL=0
MOVL C00859 V=800.0 PL=0
MOVL C00860 V=800.0 PL=0
MOVL C00861 V=800.0 PL=0
MOVL C00862 V=800.0 PL=0
MOVL C00863 V=800.0 PL=0
MOVL C00864 V=800.0 PL=0
MOVL C00865 V=800.0 PL=0
MOVL C00866 V=800.0 PL=0
MOVL C00867 V=800.0 PL=0
MOVL C00868 V=800.0 PL=0
MOVL C00869 V=800.0 PL=0
MOVL C00870 V=800.0 PL=0
MOVL C00871 V=800.0 PL=0
MOVL C00872 V=800.0 PL=0
MOVL C00873 V=800.0 PL=0
MOVL C00874 V=800.0 PL=0
MOVL C00875 V=800.0 PL=0
MOVL C00876 V=800.0 PL=0
MOVL C00877 V=800.0 PL=0
MOVL C00878 V=800.0 PL=0
MOVL C00879 V=800.0 PL=0
MOVL C00880 V=800.0 PL=0
MOVL C00881 V=800.0 PL=0
MOVL C00882 V=800.0 PL=0
MOVL C00883 V=800.0 PL=0
MOVL C00884 V=800.0 PL=0
MOVL C00885 V=800.0 PL=0
MOVL C00886 V=800.0 PL=0
MOVL C00887 V=800.0 PL=0
MOVL C00888 V=800.0 PL=0
MOVL C00889 V=800.0 PL=0
MOVL C00890 V=800.0 PL=0
MOVL C00891 V=800.0 PL=0
MOVL C00892 V=800.0 PL=0
MOVL C00893 V=800.0 PL=0
MOVL C00894 V=800.0 PL=0
MOVL C00895 V=800.0 PL=0
MOVL C00896 V=800.0 PL=0
MOVL C00897 V=800.0 PL=0
MOVL C00898 V=800.0 PL=0
MOVL C00899 V=800.0 PL=0
MOVL C00900 V=800.0 PL=0
MOVL C00901 V=800.0 PL=0
MOVL C00902 V=800.0 PL=0
MOVL C00903 V=800.0 PL=0
MOVL C00904 V=800.0 PL=0
MOVL C00905 V=800.0 PL=0
MOVL C00906 V=800.0 PL=0
MOVL C00907 V=800.0 PL=0
MOVL C00908 V=800.0 PL=0
MOVL C00909 V=800.0 PL=0
MOVL C00910 V=800.0 PL=0
MOVL C00911 V=800.0 PL=0
MOVL C00912 V=800.0 PL=0
MOVL C00913 V=800.0 PL=0
MOVL C00914 V=800.0 PL=0
MOVL C00915 V=800.0 PL=0
MOVL C00916 V=800.0 PL=0
MOVL C00917 V=800.0 PL=0
MOVL C00918 V=800.0 PL=0
MOVL C00919 V=800.0 PL=0
MOVL C00920 V=800.0 PL=0
MOVL C00921 V=800.0 PL=0
MOVL C00922 V=800.0 PL=0
MOVL C00923 V=800.0 PL=0
MOVL C00924 V=800.0 PL=0
MOVL C00925 V=800.0 PL=0
MOVL C00926 V=800.0 PL=0
MOVL C00927 V=800.0 PL=0
MOVL C00928 V=800.0 PL=0
MOVL C00929 V=800.0 PL=0
MOVL C00930 V=800.0 PL=0
MOVL C00931 V=800.0 PL=0
MOVL C00932 V=800.0 PL=0
MOVL C00933 V=800.0 PL=0
MOVL C00934 V=800.0 PL=0
MOVL C00935 V=800.0 PL=0
MOVL C00936 V=800.0 PL=0
MOVL C00937 V=800.0 PL=0
MOVL C00938 V=800.0 PL=0
MOVL C00939 V=800.0 PL=0
MOVL C00940 V=800.0 PL=0
MOVL C00941 V=800.0 PL=0
MOVL C00942 V=800.0 PL=0
MOVL C00943 V=800.0 PL=0
MOVL C00944 V=800.0 PL=0
MOVL C00945 V=800.0 PL=0
MOVL C00946 V=800.0 PL=0
MOVL C00947 V=800.0 PL=0
MOVL C00948 V=800.0 PL=0
MOVL C00949 V=800.0 PL=0
MOVL C00950 V=800.0 PL=0
MOVL C00951 V=800.0 PL=0
MOVL C00952 V=800.0 PL=0
MOVL C00953 V=800.0 PL=0
MOVL C00954 V=800.0 PL=0
MOVL C00955 V=800.0 PL=0
MOVL C00956 V=800.0 PL=0
MOVL C00957 V=800.0 PL=0
MOVL C00958 V=800.0 PL=0
MOVL C00959 V=800.0 PL=0
MOVL C00960 V=800.0 PL=0
MOVL C00961 V=800.0 PL=0
MOVL C00962 V=800.0 PL=0
MOVL C00963 V=800.0 PL=0
MOVL C00964 V=800.0 PL=0
MOVL C00965 V=800.0 PL=0
MOVL C00966 V=800.0 PL=0
MOVL C00967 V=800.0 PL=0
MOVL C00968 V=800.0 PL=0
MOVL C00969 V=800.0 PL=0
MOVL C00970 V=800.0 PL=0
MOVL C00971 V=800.0 PL=0
MOVL C00972 V=800.0 PL=0
MOVL C00973 V=800.0 PL=0
MOVL C00974 V=800.0 PL=0
MOVL C00975 V=800.0 PL=0
MOVL C00976 V=800.0 PL=0
MOVL C00977 V=800.0 PL=0
MOVL C00978 V=800.0 PL=0
MOVL C00979 V=800.0 PL=0
MOVL C00980 V=800.0 PL=0
MOVL C00981 V=800.0 PL=0
MOVL C00982 V=800.0 PL=0
MOVL C00983 V=800.0 PL=0
MOVL C00984 V=800.0 PL=0
MOVL C00985 V=800.0 PL=0
MOVL C00986 V=800.0 PL=0
MOVL C00987 V=800.0 PL=0
MOVL C00988 V=800.0 PL=0
MOVL C00989 V=800.0 PL=0
MOVL C00990 V=800.0 PL=0
MOVL C00991 V=800.0 PL=0
MOVL C00992 V=800.0 PL=0
MOVL C00993 V=800.0 PL=0
MOVL C00994 V=800.0 PL=0
MOVL C00995 V=800.0 PL=0
MOVL C00996 V=800.0 PL=0
MOVL C00997 V=800.0 PL=0
MOVL C00998 V=800.0 PL=0
MOVL C00999 V=800.0 PL=0
MOVL C01000 V=800.0 PL=0
MOVL C01001 V=800.0 PL=0
MOVL C01002 V=800.0 PL=0
MOVL C01003 V=800.0 PL=0
MOVL C01004 V=800.0 PL=0
MOVL C01005 V=800.0 PL=0
MOVL C01006 V=800.0 PL=0
MOVL C01007 V=800.0 PL=0
MOVL C01008 V=800.0 PL=0
MOVL C01009 V=800.0 PL=0
MOVL C01010 V=800.0 PL=0
MOVL C01011 V=800.0 PL=0
MOVL C01012 V=800.0 PL=0
MOVL C01013 V=800.0 PL=0
MOVL C01014 V=800.0 PL=0
MOVL C01015 V=800.0 PL=0
MOVL C01016 V=800.0 PL=0
MOVL C01017 V=800.0 PL=0
MOVL C01018 V=800.0 PL=0
MOVL C01019 V=800.0 PL=0
MOVL C01020 V=800.0 PL=0
MOVL C01021 V=800.0 PL=0
MOVL C01022 V=800.0 PL=0
MOVL C01023 V=800.0 PL=0
MOVL C01024 V=800.0 PL=0
MOVL C01025 V=800.0 PL=0
MOVL C01026 V=800.0 PL=0
MOVL C01027 V=800.0 PL=0
MOVL C01028 V=800.0 PL=0
MOVL C01029 V=800.0 PL=0
MOVL C01030 V=800.0 PL=0
MOVL C01031 V=800.0 PL=0
MOVL C01032 V=800.0 PL=0
MOVL C01033 V=800.0 PL=0
MOVL C01034 V=800.0 PL=0
MOVL C01035 V=800.0 PL=0
MOVL C01036 V=800.0 PL=0
MOVL C01037 V=800.0 PL=0
MOVL C01038 V=800.0 PL=0
MOVL C01039 V=800.0 PL=0
MOVL C01040 V=800.0 PL=0
MOVL C01041 V=800.0 PL=0
MOVL C01042 V=800.0 PL=0
MOVL C01043 V=800.0 PL=0
MOVL C01044 V=800.0 PL=0
MOVL C01045 V=800.0 PL=0
MOVL C01046 V=800.0 PL=0
MOVL C01047 V=800.0 PL=0
MOVL C01048 V=800.0 PL=0
MOVL C01049 V=800.0 PL=0
MOVL C01050 V=800.0 PL=0
MOVL C01051 V=800.0 PL=0
MOVL C01052 V=800.0 PL=0
MOVL C01053 V=800.0 PL=0
MOVL C01054 V=800.0 PL=0
MOVL C01055 V=800.0 PL=0
MOVL C01056 V=800.0 PL=0
MOVL C01057 V=800.0 PL=0
MOVL C01058 V=800.0 PL=0
MOVL C01059 V=800.0 PL=0
MOVL C01060 V=800.0 PL=0
MOVL C01061 V=800.0 PL=0
MOVL C01062 V=800.0 PL=0
MOVL C01063 V=800.0 PL=0
MOVL C01064 V=800.0 PL=0
MOVL C01065 V=800.0 PL=0
MOVL C01066 V=800.0 PL=0
MOVL C01067 V=800.0 PL=0
MOVL C01068 V=800.0 PL=0
MOVL C01069 V=800.0 PL=0
MOVL C01070 V=800.0 PL=0
MOVL C01071 V=800.0 PL=0
MOVL C01072 V=800.0 PL=0
MOVL C01073 V=800.0 PL=0
MOVL C01074 V=800.0 PL=0
MOVL C01075 V=800.0 PL=0
MOVL C01076 V=800.0 PL=0
MOVL C01077 V=800.0 PL=0
MOVL C01078 V=800.0 PL=0
MOVL C01079 V=800.0 PL=0
MOVL C01080 V=800.0 PL=0
MOVL C01081 V=800.0 PL=0
MOVL C01082 V=800.0 PL=0
MOVL C01083 V=800.0 PL=0
MOVL C01084 V=800.0 PL=0
MOVL C01085 V=800.0 PL=0
MOVL C01086 V=800.0 PL=0
MOVL C01087 V=800.0 PL=0
MOVL C01088 V=800.0 PL=0
MOVL C01089 V=800.0 PL=0
MOVL C01090 V=800.0 PL=0
MOVL C01091 V=800.0 PL=0
MOVL C01092 V=800.0 PL=0
MOVL C01093 V=800.0 PL=0
MOVL C01094 V=800.0 PL=0
MOVL C01095 V=800.0 PL=0
MOVL C01096 V=800.0 PL=0
MOVL C01097 V=800.0 PL=0
MOVL C01098 V=800.0 PL=0
MOVL C01099 V=800.0 PL=0
MOVL C01100 V=800.0 PL=0
MOVL C01101 V=800.0 PL=0
MOVL C01102 V=800.0 PL=0
MOVL C01103 V=800.0 PL=0
MOVL C01104 V=800.0 PL=0
MOVL C01105 V=800.0 PL=0
MOVL C01106 V=800.0 PL=0
MOVL C01107 V=800.0 PL=0
MOVL C01108 V=800.0 PL=0
MOVL C01109 V=800.0 PL=0
MOVL C01110 V=800.0 PL=0
MOVL C01111 V=800.0 PL=0
MOVL C01112 V=800.0 PL=0
MOVL C01113 V=800.0 PL=0
MOVL C01114 V=800.0 PL=0
MOVL C01115 V=800.0 PL=0
MOVL C01116 V=800.0 PL=0
MOVL C01117 V=800.0 PL=0
MOVL C01118 V=800.0 PL=0
MOVL C01119 V=800.0 PL=0
MOVL C01120 V=800.0 PL=0
MOVL C01121 V=800.0 PL=0
MOVL C01122 V=800.0 PL=0
MOVL C01123 V=800.0 PL=0
MOVL C01124 V=800.0 PL=0
MOVL C01125 V=800.0 PL=0
MOVL C01126 V=800.0 PL=0
MOVL C01127 V=800.0 PL=0
MOVL C01128 V=800.0 PL=0
MOVL C01129 V=800.0 PL=0
MOVL C01130 V=800.0 PL=0
MOVL C01131 V=800.0 PL=0
MOVL C01132 V=800.0 PL=0
MOVL C01133 V=800.0 PL=0
MOVL C01134 V=800.0 PL=0
MOVL C01135 V=800.0 PL=0
MOVL C01136 V=800.0 PL=0
MOVL C01137 V=800.0 PL=0
MOVL C01138 V=800.0 PL=0
MOVL C01139 V=800.0 PL=0
MOVL C01140 V=800.0 PL=0
MOVL C01141 V=800.0 PL=0
MOVL C01142 V=800.0 PL=0
MOVL C01143 V=800.0 PL=0
MOVL C01144 V=800.0 PL=0
MOVL C01145 V=800.0 PL=0
MOVL C01146 V=800.0 PL=0
MOVL C01147 V=800.0 PL=0
MOVL C01148 V=800.0 PL=0
MOVL C01149 V=800.0 PL=0
MOVL C01150 V=800.0 PL=0
MOVL C01151 V=800.0 PL=0
MOVL C01152 V=800.0 PL=0
MOVL C01153 V=800.0 PL=0
MOVL C01154 V=800.0 PL=0
MOVL C01155 V=800.0 PL=0
MOVL C01156 V=800.0 PL=0
MOVL C01157 V=800.0 PL=0
MOVL C01158 V=800.0 PL=0
MOVL C01159 V=800.0 PL=0
MOVL C01160 V=800.0 PL=0
MOVL C01161 V=800.0 PL=0
MOVL C01162 V=800.0 PL=0
MOVL C01163 V=800.0 PL=0
MOVL C01164 V=800.0 PL=0
MOVL C01165 V=800.0 PL=0
MOVL C01166 V=800.0 PL=0
MOVL C01167 V=800.0 PL=0
MOVL C01168 V=800.0 PL=0
MOVL C01169 V=800.0 PL=0
MOVL C01170 V=800.0 PL=0
MOVL C01171 V=800.0 PL=0
MOVL C01172 V=800.0 PL=0
MOVL C01173 V=800.0 PL=0
MOVL C01174 V=800.0 PL=0
MOVL C01175 V=800.0 PL=0
MOVL C01176 V=800.0 PL=0
MOVL C01177 V=800.0 PL=0
MOVL C01178 V=800.0 PL=0
MOVL C01179 V=800.0 PL=0
MOVL C01180 V=800.0 PL=0
MOVL C01181 V=800.0 PL=0
MOVL C01182 V=800.0 PL=0
MOVL C01183 V=800.0 PL=0
MOVL C01184 V=800.0 PL=0
MOVL C01185 V=800.0 PL=0
MOVL C01186 V=800.0 PL=0
MOVL C01187 V=800.0 PL=0
MOVL C01188 V=800.0 PL=0
MOVL C01189 V=800.0 PL=0
MOVL C01190 V=800.0 PL=0
MOVL C01191 V=800.0 PL=0
MOVL C01192 V=800.0 PL=0
MOVL C01193 V=800.0 PL=0
MOVL C01194 V=800.0 PL=0
MOVL C01195 V=800.0 PL=0
MOVL C01196 V=800.0 PL=0
MOVL C01197 V=800.0 PL=0
MOVL C01198 V=800.0 PL=0
MOVL C01199 V=800.0 PL=0
MOVL C01200 V=800.0 PL=0
MOVL C01201 V=800.0 PL=0
MOVL C01202 V=800.0 PL=0
MOVL C01203 V=800.0 PL=0
MOVL C01204 V=800.0 PL=0
MOVL C01205 V=800.0 PL=0
MOVL C01206 V=800.0 PL=0
MOVL C01207 V=800.0 PL=0
MOVL C01208 V=800.0 PL=0
MOVL C01209 V=800.0 PL=0
MOVL C01210 V=800.0 PL=0
MOVL C01211 V=800.0 PL=0
MOVL C01212 V=800.0 PL=0
MOVL C01213 V=800.0 PL=0
MOVL C01214 V=800.0 PL=0
MOVL C01215 V=800.0 PL=0
MOVL C01216 V=800.0 PL=0
MOVL C01217 V=800.0 PL=0
MOVL C01218 V=800.0 PL=0
MOVL C01219 V=800.0 PL=0
MOVL C01220 V=800.0 PL=0
MOVL C01221 V=800.0 PL=0
MOVL C01222 V=800.0 PL=0
MOVL C01223 V=800.0 PL=0
MOVL C01224 V=800.0 PL=0
MOVL C01225 V=800.0 PL=0
MOVL C01226 V=800.0 PL=0
MOVL C01227 V=800.0 PL=0
MOVL C01228 V=800.0 PL=0
MOVL C01229 V=800.0 PL=0
MOVL C01230 V=800.0 PL=0
MOVL C01231 V=800.0 PL=0
MOVL C01232 V=800.0 PL=0
MOVL C01233 V=800.0 PL=0
MOVL C01234 V=800.0 PL=0
MOVL C01235 V=800.0 PL=0
MOVL C01236 V=800.0 PL=0
MOVL C01237 V=800.0 PL=0
MOVL C01238 V=800.0 PL=0
MOVL C01239 V=800.0 PL=0
MOVL C01240 V=800.0 PL=0
MOVL C01241 V=800.0 PL=0
MOVL C01242 V=800.0 PL=0
MOVL C01243 V=800.0 PL=0
MOVL C01244 V=800.0 PL=0
MOVL C01245 V=800.0 PL=0
MOVL C01246 V=800.0 PL=0
MOVL C01247 V=800.0 PL=0
MOVL C01248 V=800.0 PL=0
MOVL C01249 V=800.0 PL=0
MOVL C01250 V=800.0 PL=0
MOVL C01251 V=800.0 PL=0
MOVL C01252 V=800.0 PL=0
MOVL C01253 V=800.0 PL=0
MOVL C01254 V=800.0 PL=0
MOVL C01255 V=800.0 PL=0
MOVL C01256 V=800.0 PL=0
MOVL C01257 V=800.0 PL=0
MOVL C01258 V=800.0 PL=0
MOVL C01259 V=800.0 PL=0
MOVL C01260 V=800.0 PL=0
MOVL C01261 V=800.0 PL=0
MOVL C01262 V=800.0 PL=0
MOVL C01263 V=800.0 PL=0
MOVL C01264 V=800.0 PL=0
MOVL C01265 V=800.0 PL=0
MOVL C01266 V=800.0 PL=0
MOVL C01267 V=800.0 PL=0
MOVL C01268 V=800.0 PL=0
MOVL C01269 V=800.0 PL=0
MOVL C01270 V=800.0 PL=0
MOVL C01271 V=800.0 PL=0
MOVL C01272 V=800.0 PL=0
MOVL C01273 V=800.0 PL=0
MOVL C01274 V=800.0 PL=0
MOVL C01275 V=800.0 PL=0
MOVL C01276 V=800.0 PL=0
MOVL C01277 V=800.0 PL=0
MOVL C01278 V=800.0 PL=0
MOVL C01279 V=800.0 PL=0
MOVL C01280 V=800.0 PL=0
MOVL C01281 V=800.0 PL=0
MOVL C01282 V=800.0 PL=0
MOVL C01283 V=800.0 PL=0
MOVL C01284 V=800.0 PL=0
MOVL C01285 V=800.0 PL=0
MOVL C01286 V=800.0 PL=0
MOVL C01287 V=800.0 PL=0
MOVL C01288 V=800.0 PL=0
MOVL C01289 V=800.0 PL=0
MOVL C01290 V=800.0 PL=0
MOVL C01291 V=800.0 PL=0
MOVL C01292 V=800.0 PL=0
MOVL C01293 V=800.0 PL=0
MOVL C01294 V=800.0 PL=0
MOVL C01295 V=800.0 PL=0
MOVL C01296 V=800.0 PL=0
MOVL C01297 V=800.0 PL=0
MOVL C01298 V=800.0 PL=0
MOVL C01299 V=800.0 PL=0
MOVL C01300 V=800.0 PL=0
MOVL C01301 V=800.0 PL=0
MOVL C01302 V=800.0 PL=0
MOVL C01303 V=800.0 PL=0
MOVL C01304 V=800.0 PL=0
MOVL C01305 V=800.0 PL=0
MOVL C01306 V=800.0 PL=0
MOVL C01307 V=800.0 PL=0
MOVL C01308 V=800.0 PL=0
MOVL C01309 V=800.0 PL=0
MOVL C01310 V=800.0 PL=0
MOVL C01311 V=800.0 PL=0
MOVL C01312 V=800.0 PL=0
MOVL C01313 V=800.0 PL=0
MOVL C01314 V=800.0 PL=0
MOVL C01315 V=800.0 PL=0
MOVL C01316 V=800.0 PL=0
MOVL C01317 V=800.0 PL=0
MOVL C01318 V=800.0 PL=0
MOVL C01319 V=800.0 PL=0
MOVL C01320 V=800.0 PL=0
MOVL C01321 V=800.0 PL=0
MOVL C01322 V=800.0 PL=0
MOVL C01323 V=800.0 PL=0
MOVL C01324 V=800.0 PL=0
MOVL C01325 V=800.0 PL=0
MOVL C01326 V=800.0 PL=0
MOVL C01327 V=800.0 PL=0
MOVL C01328 V=800.0 PL=0
MOVL C01329 V=800.0 PL=0
MOVL C01330 V=800.0 PL=0
MOVL C01331 V=800.0 PL=0
MOVL C01332 V=800.0 PL=0
MOVL C01333 V=800.0 PL=0
MOVL C01334 V=800.0 PL=0
MOVL C01335 V=800.0 PL=0
MOVL C01336 V=800.0 PL=0
MOVL C01337 V=800.0 PL=0
MOVL C01338 V=800.0 PL=0
MOVL C01339 V=800.0 PL=0
MOVL C01340 V=800.0 PL=0
MOVL C01341 V=800.0 PL=0
MOVL C01342 V=800.0 PL=0
MOVL C01343 V=800.0 PL=0
MOVL C01344 V=800.0 PL=0
MOVL C01345 V=800.0 PL=0
MOVL C01346 V=800.0 PL=0
MOVL C01347 V=800.0 PL=0
MOVL C01348 V=800.0 PL=0
MOVL C01349 V=800.0 PL=0
MOVL C01350 V=800.0 PL=0
MOVL C01351 V=800.0 PL=0
MOVL C01352 V=800.0 PL=0
MOVL C01353 V=800.0 PL=0
MOVL C01354 V=800.0 PL=0
MOVL C01355 V=800.0 PL=0
MOVL C01356 V=800.0 PL=0
MOVL C01357 V=800.0 PL=0
MOVL C01358 V=800.0 PL=0
MOVL C01359 V=800.0 PL=0
MOVL C01360 V=800.0 PL=0
MOVL C01361 V=800.0 PL=0
MOVL C01362 V=800.0 PL=0
MOVL C01363 V=800.0 PL=0
MOVL C01364 V=800.0 PL=0
MOVL C01365 V=800.0 PL=0
MOVL C01366 V=800.0 PL=0
MOVL C01367 V=800.0 PL=0
MOVL C01368 V=800.0 PL=0
MOVL C01369 V=800.0 PL=0
MOVL C01370 V=800.0 PL=0
MOVL C01371 V=800.0 PL=0
MOVL C01372 V=800.0 PL=0
MOVL C01373 V=800.0 PL=0
MOVL C01374 V=800.0 PL=0
MOVL C01375 V=800.0 PL=0
MOVL C01376 V=800.0 PL=0
MOVL C01377 V=800.0 PL=0
MOVL C01378 V=800.0 PL=0
MOVL C01379 V=800.0 PL=0
MOVL C01380 V=800.0 PL=0
MOVL C01381 V=800.0 PL=0
MOVL C01382 V=800.0 PL=0
MOVL C01383 V=800.0 PL=0
MOVL C01384 V=800.0 PL=0
MOVL C01385 V=800.0 PL=0
MOVL C01386 V=800.0 PL=0
MOVL C01387 V=800.0 PL=0
MOVL C01388 V=800.0 PL=0
MOVL C01389 V=800.0 PL=0
MOVL C01390 V=800.0 PL=0
MOVL C01391 V=800.0 PL=0
MOVL C01392 V=800.0 PL=0
MOVL C01393 V=800.0 PL=0
MOVL C01394 V=800.0 PL=0
MOVL C01395 V=800.0 PL=0
MOVL C01396 V=800.0 PL=0
MOVL C01397 V=800.0 PL=0
MOVL C01398 V=800.0 PL=0
MOVL C01399 V=800.0 PL=0
MOVL C01400 V=800.0 PL=0
MOVL C01401 V=800.0 PL=0
MOVL C01402 V=800.0 PL=0
MOVL C01403 V=800.0 PL=0
MOVL C01404 V=800.0 PL=0
MOVL C01405 V=800.0 PL=0
MOVL C01406 V=800.0 PL=0
MOVL C01407 V=800.0 PL=0
MOVL C01408 V=800.0 PL=0
MOVL C01409 V=800.0 PL=0
MOVL C01410 V=800.0 PL=0
MOVL C01411 V=800.0 PL=0
MOVL C01412 V=800.0 PL=0
MOVL C01413 V=800.0 PL=0
MOVL C01414 V=800.0 PL=0
MOVL C01415 V=800.0 PL=0
MOVL C01416 V=800.0 PL=0
MOVL C01417 V=800.0 PL=0
MOVL C01418 V=800.0 PL=0
MOVL C01419 V=800.0 PL=0
MOVL C01420 V=800.0 PL=0
MOVL C01421 V=800.0 PL=0
MOVL C01422 V=800.0 PL=0
MOVL C01423 V=800.0 PL=0
MOVL C01424 V=800.0 PL=0
MOVL C01425 V=800.0 PL=0
MOVL C01426 V=800.0 PL=0
MOVL C01427 V=800.0 PL=0
MOVL C01428 V=800.0 PL=0
MOVL C01429 V=800.0 PL=0
MOVL C01430 V=800.0 PL=0
MOVL C01431 V=800.0 PL=0
MOVL C01432 V=800.0 PL=0
MOVL C01433 V=800.0 PL=0
MOVL C01434 V=800.0 PL=0
MOVL C01435 V=800.0 PL=0
MOVL C01436 V=800.0 PL=0
MOVL C01437 V=800.0 PL=0
MOVL C01438 V=800.0 PL=0
MOVL C01439 V=800.0 PL=0
MOVL C01440 V=800.0 PL=0
MOVL C01441 V=800.0 PL=0
MOVL C01442 V=800.0 PL=0
MOVL C01443 V=800.0 PL=0
MOVL C01444 V=800.0 PL=0
MOVL C01445 V=800.0 PL=0
MOVL C01446 V=800.0 PL=0
MOVL C01447 V=800.0 PL=0
MOVL C01448 V=800.0 PL=0
MOVL C01449 V=800.0 PL=0
MOVL C01450 V=800.0 PL=0
MOVL C01451 V=800.0 PL=0
MOVL C01452 V=800.0 PL=0
MOVL C01453 V=800.0 PL=0
MOVL C01454 V=800.0 PL=0
MOVL C01455 V=800.0 PL=0
MOVL C01456 V=800.0 PL=0
MOVL C01457 V=800.0 PL=0
MOVL C01458 V=800.0 PL=0
MOVL C01459 V=800.0 PL=0
MOVL C01460 V=800.0 PL=0
MOVL C01461 V=800.0 PL=0
MOVL C01462 V=800.0 PL=0
MOVL C01463 V=800.0 PL=0
MOVL C01464 V=800.0 PL=0
MOVL C01465 V=800.0 PL=0
MOVL C01466 V=800.0 PL=0
MOVL C01467 V=800.0 PL=0
MOVL C01468 V=800.0 PL=0
MOVL C01469 V=800.0 PL=0
MOVL C01470 V=800.0 PL=0
MOVL C01471 V=800.0 PL=0
MOVL C01472 V=800.0 PL=0
MOVL C01473 V=800.0 PL=0
MOVL C01474 V=800.0 PL=0
MOVL C01475 V=800.0 PL=0
MOVL C01476 V=800.0 PL=0
MOVL C01477 V=800.0 PL=0
MOVL C01478 V=800.0 PL=0
MOVL C01479 V=800.0 PL=0
MOVL C01480 V=800.0 PL=0
MOVL C01481 V=800.0 PL=0
MOVL C01482 V=800.0 PL=0
MOVL C01483 V=800.0 PL=0
MOVL C01484 V=800.0 PL=0
MOVL C01485 V=800.0 PL=0
MOVL C01486 V=800.0 PL=0
MOVL C01487 V=800.0 PL=0
MOVL C01488 V=800.0 PL=0
MOVL C01489 V=800.0 PL=0
MOVL C01490 V=800.0 PL=0
MOVL C01491 V=800.0 PL=0
MOVL C01492 V=800.0 PL=0
MOVL C01493 V=800.0 PL=0
MOVL C01494 V=800.0 PL=0
MOVL C01495 V=800.0 PL=0
MOVL C01496 V=800.0 PL=0
MOVL C01497 V=800.0 PL=0
MOVL C01498 V=800.0 PL=0
MOVL C01499 V=800.0 PL=0
MOVL C01500 V=800.0 PL=0
MOVL C01501 V=800.0 PL=0
MOVL C01502 V=800.0 PL=0
MOVL C01503 V=800.0 PL=0
MOVL C01504 V=800.0 PL=0
MOVL C01505 V=800.0 PL=0
MOVL C01506 V=800.0 PL=0
MOVL C01507 V=800.0 PL=0
MOVL C01508 V=800.0 PL=0
MOVL C01509 V=800.0 PL=0
MOVL C01510 V=800.0 PL=0
MOVL C01511 V=800.0 PL=0
MOVL C01512 V=800.0 PL=0
MOVL C01513 V=800.0 PL=0
MOVL C01514 V=800.0 PL=0
MOVL C01515 V=800.0 PL=0
MOVL C01516 V=800.0 PL=0
MOVL C01517 V=800.0 PL=0
MOVL C01518 V=800.0 PL=0
MOVL C01519 V=800.0 PL=0
MOVL C01520 V=800.0 PL=0
MOVL C01521 V=800.0 PL=0
MOVL C01522 V=800.0 PL=0
MOVL C01523 V=800.0 PL=0
MOVL C01524 V=800.0 PL=0
MOVL C01525 V=800.0 PL=0
MOVL C01526 V=800.0 PL=0
MOVL C01527 V=800.0 PL=0
MOVL C01528 V=800.0 PL=0
MOVL C01529 V=800.0 PL=0
MOVL C01530 V=800.0 PL=0
MOVL C01531 V=800.0 PL=0
MOVL C01532 V=800.0 PL=0
MOVL C01533 V=800.0 PL=0
MOVL C01534 V=800.0 PL=0
MOVL C01535 V=800.0 PL=0
MOVL C01536 V=800.0 PL=0
MOVL C01537 V=800.0 PL=0
MOVL C01538 V=800.0 PL=0
MOVL C01539 V=800.0 PL=0
MOVL C01540 V=800.0 PL=0
MOVL C01541 V=800.0 PL=0
MOVL C01542 V=800.0 PL=0
MOVL C01543 V=800.0 PL=0
MOVL C01544 V=800.0 PL=0
MOVL C01545 V=800.0 PL=0
MOVL C01546 V=800.0 PL=0
MOVL C01547 V=800.0 PL=0
MOVL C01548 V=800.0 PL=0
MOVL C01549 V=800.0 PL=0
MOVL C01550 V=800.0 PL=0
MOVL C01551 V=800.0 PL=0
MOVL C01552 V=800.0 PL=0
MOVL C01553 V=800.0 PL=0
MOVL C01554 V=800.0 PL=0
MOVL C01555 V=800.0 PL=0
MOVL C01556 V=800.0 PL=0
MOVL C01557 V=800.0 PL=0
MOVL C01558 V=800.0 PL=0
MOVL C01559 V=800.0 PL=0
MOVL C01560 V=800.0 PL=0
MOVL C01561 V=800.0 PL=0
MOVL C01562 V=800.0 PL=0
MOVL C01563 V=800.0 PL=0
MOVL C01564 V=800.0 PL=0
MOVL C01565 V=800.0 PL=0
MOVL C01566 V=800.0 PL=0
MOVL C01567 V=800.0 PL=0
MOVL C01568 V=800.0 PL=0
MOVL C01569 V=800.0 PL=0
MOVL C01570 V=800.0 PL=0
MOVL C01571 V=800.0 PL=0
MOVL C01572 V=800.0 PL=0
MOVL C01573 V=800.0 PL=0
MOVL C01574 V=800.0 PL=0
MOVL C01575 V=800.0 PL=0
MOVL C01576 V=800.0 PL=0
MOVL C01577 V=800.0 PL=0
MOVL C01578 V=800.0 PL=0
MOVL C01579 V=800.0 PL=0
MOVL C01580 V=800.0 PL=0
MOVL C01581 V=800.0 PL=0
MOVL C01582 V=800.0 PL=0
MOVL C01583 V=800.0 PL=0
MOVL C01584 V=800.0 PL=0
MOVL C01585 V=800.0 PL=0
MOVL C01586 V=800.0 PL=0
MOVL C01587 V=800.0 PL=0
MOVL C01588 V=800.0 PL=0
MOVL C01589 V=800.0 PL=0
MOVL C01590 V=800.0 PL=0
MOVL C01591 V=800.0 PL=0
MOVL C01592 V=800.0 PL=0
MOVL C01593 V=800.0 PL=0
MOVL C01594 V=800.0 PL=0
MOVL C01595 V=800.0 PL=0
MOVL C01596 V=800.0 PL=0
MOVL C01597 V=800.0 PL=0
MOVL C01598 V=800.0 PL=0
MOVL C01599 V=800.0 PL=0
MOVL C01600 V=800.0 PL=0
MOVL C01601 V=800.0 PL=0
MOVL C01602 V=800.0 PL=0
MOVL C01603 V=800.0 PL=0
MOVL C01604 V=800.0 PL=0
MOVL C01605 V=800.0 PL=0
MOVL C01606 V=800.0 PL=0
MOVL C01607 V=800.0 PL=0
MOVL C01608 V=800.0 PL=0
MOVL C01609 V=800.0 PL=0
MOVL C01610 V=800.0 PL=0
MOVL C01611 V=800.0 PL=0
MOVL C01612 V=800.0 PL=0
MOVL C01613 V=800.0 PL=0
MOVL C01614 V=800.0 PL=0
MOVL C01615 V=800.0 PL=0
MOVL C01616 V=800.0 PL=0
MOVL C01617 V=800.0 PL=0
MOVL C01618 V=800.0 PL=0
MOVL C01619 V=800.0 PL=0
MOVL C01620 V=800.0 PL=0
MOVL C01621 V=800.0 PL=0
MOVL C01622 V=800.0 PL=0
MOVL C01623 V=800.0 PL=0
MOVL C01624 V=800.0 PL=0
MOVL C01625 V=800.0 PL=0
MOVL C01626 V=800.0 PL=0
MOVL C01627 V=800.0 PL=0
MOVL C01628 V=800.0 PL=0
MOVL C01629 V=800.0 PL=0
MOVL C01630 V=800.0 PL=0
MOVL C01631 V=800.0 PL=0
MOVL C01632 V=800.0 PL=0
MOVL C01633 V=800.0 PL=0
MOVL C01634 V=800.0 PL=0
MOVL C01635 V=800.0 PL=0
MOVL C01636 V=800.0 PL=0
MOVL C01637 V=800.0 PL=0
MOVL C01638 V=800.0 PL=0
MOVL C01639 V=800.0 PL=0
MOVL C01640 V=800.0 PL=0
MOVL C01641 V=800.0 PL=0
MOVL C01642 V=800.0 PL=0
MOVL C01643 V=800.0 PL=0
MOVL C01644 V=800.0 PL=0
MOVL C01645 V=800.0 PL=0
MOVL C01646 V=800.0 PL=0
MOVL C01647 V=800.0 PL=0
MOVL C01648 V=800.0 PL=0
MOVL C01649 V=800.0 PL=0
MOVL C01650 V=800.0 PL=0
MOVL C01651 V=800.0 PL=0
MOVL C01652 V=800.0 PL=0
MOVL C01653 V=800.0 PL=0
MOVL C01654 V=800.0 PL=0
MOVL C01655 V=800.0 PL=0
MOVL C01656 V=800.0 PL=0
MOVL C01657 V=800.0 PL=0
MOVL C01658 V=800.0 PL=0
MOVL C01659 V=800.0 PL=0
MOVL C01660 V=800.0 PL=0
MOVL C01661 V=800.0 PL=0
MOVL C01662 V=800.0 PL=0
MOVL C01663 V=800.0 PL=0
MOVL C01664 V=800.0 PL=0
MOVL C01665 V=800.0 PL=0
MOVL C01666 V=800.0 PL=0
MOVL C01667 V=800.0 PL=0
MOVL C01668 V=800.0 PL=0
MOVL C01669 V=800.0 PL=0
MOVL C01670 V=800.0 PL=0
MOVL C01671 V=800.0 PL=0
MOVL C01672 V=800.0 PL=0
MOVL C01673 V=800.0 PL=0
MOVL C01674 V=800.0 PL=0
MOVL C01675 V=800.0 PL=0
MOVL C01676 V=800.0 PL=0
MOVL C01677 V=800.0 PL=0
MOVL C01678 V=800.0 PL=0
MOVL C01679 V=800.0 PL=0
MOVL C01680 V=800.0 PL=0
MOVL C01681 V=800.0 PL=0
MOVL C01682 V=800.0 PL=0
MOVL C01683 V=800.0 PL=0
MOVL C01684 V=800.0 PL=0
MOVL C01685 V=800.0 PL=0
MOVL C01686 V=800.0 PL=0
MOVL C01687 V=800.0 PL=0
MOVL C01688 V=800.0 PL=0
MOVL C01689 V=800.0 PL=0
MOVL C01690 V=800.0 PL=0
MOVL C01691 V=800.0 PL=0
MOVL C01692 V=800.0 PL=0
MOVL C01693 V=800.0 PL=0
MOVL C01694 V=800.0 PL=0
MOVL C01695 V=800.0 PL=0
MOVL C01696 V=800.0 PL=0
MOVL C01697 V=800.0 PL=0
MOVL C01698 V=800.0 PL=0
MOVL C01699 V=800.0 PL=0
MOVL C01700 V=800.0 PL=0
MOVL C01701 V=800.0 PL=0
MOVL C01702 V=800.0 PL=0
MOVL C01703 V=800.0 PL=0
MOVL C01704 V=800.0 PL=0
MOVL C01705 V=800.0 PL=0
MOVL C01706 V=800.0 PL=0
MOVL C01707 V=800.0 PL=0
MOVL C01708 V=800.0 PL=0
MOVL C01709 V=800.0 PL=0
MOVL C01710 V=800.0 PL=0
MOVL C01711 V=800.0 PL=0
MOVL C01712 V=800.0 PL=0
MOVL C01713 V=800.0 PL=0
MOVL C01714 V=800.0 PL=0
MOVL C01715 V=800.0 PL=0
MOVL C01716 V=800.0 PL=0
MOVL C01717 V=800.0 PL=0
MOVL C01718 V=800.0 PL=0
MOVL C01719 V=800.0 PL=0
MOVL C01720 V=800.0 PL=0
MOVL C01721 V=800.0 PL=0
MOVL C01722 V=800.0 PL=0
MOVL C01723 V=800.0 PL=0
MOVL C01724 V=800.0 PL=0
MOVL C01725 V=800.0 PL=0
MOVL C01726 V=800.0 PL=0
MOVL C01727 V=800.0 PL=0
MOVL C01728 V=800.0 PL=0
MOVL C01729 V=800.0 PL=0
MOVL C01730 V=800.0 PL=0
MOVL C01731 V=800.0 PL=0
MOVL C01732 V=800.0 PL=0
MOVL C01733 V=800.0 PL=0
MOVL C01734 V=800.0 PL=0
MOVL C01735 V=800.0 PL=0
MOVL C01736 V=800.0 PL=0
MOVL C01737 V=800.0 PL=0
MOVL C01738 V=800.0 PL=0
MOVL C01739 V=800.0 PL=0
MOVL C01740 V=800.0 PL=0
MOVL C01741 V=800.0 PL=0
MOVL C01742 V=800.0 PL=0
MOVL C01743 V=800.0 PL=0
MOVL C01744 V=800.0 PL=0
MOVL C01745 V=800.0 PL=0
MOVL C01746 V=800.0 PL=0
MOVL C01747 V=800.0 PL=0
MOVL C01748 V=800.0 PL=0
MOVL C01749 V=800.0 PL=0
MOVL C01750 V=800.0 PL=0
MOVL C01751 V=800.0 PL=0
MOVL C01752 V=800.0 PL=0
MOVL C01753 V=800.0 PL=0
MOVL C01754 V=800.0 PL=0
MOVL C01755 V=800.0 PL=0
MOVL C01756 V=800.0 PL=0
MOVL C01757 V=800.0 PL=0
MOVL C01758 V=800.0 PL=0
MOVL C01759 V=800.0 PL=0
MOVL C01760 V=800.0 PL=0
MOVL C01761 V=800.0 PL=0
MOVL C01762 V=800.0 PL=0
MOVL C01763 V=800.0 PL=0
MOVL C01764 V=800.0 PL=0
MOVL C01765 V=800.0 PL=0
MOVL C01766 V=800.0 PL=0
MOVL C01767 V=800.0 PL=0
MOVL C01768 V=800.0 PL=0
MOVL C01769 V=800.0 PL=0
MOVL C01770 V=800.0 PL=0
MOVL C01771 V=800.0 PL=0
MOVL C01772 V=800.0 PL=0
MOVL C01773 V=800.0 PL=0
MOVL C01774 V=800.0 PL=0
MOVL C01775 V=800.0 PL=0
MOVL C01776 V=800.0 PL=0
MOVL C01777 V=800.0 PL=0
MOVL C01778 V=800.0 PL=0
MOVL C01779 V=800.0 PL=0
MOVL C01780 V=800.0 PL=0
MOVL C01781 V=800.0 PL=0
MOVL C01782 V=800.0 PL=0
MOVL C01783 V=800.0 PL=0
MOVL C01784 V=800.0 PL=0
MOVL C01785 V=800.0 PL=0
MOVL C01786 V=800.0 PL=0
MOVL C01787 V=800.0 PL=0
MOVL C01788 V=800.0 PL=0
MOVL C01789 V=800.0 PL=0
MOVL C01790 V=800.0 PL=0
MOVL C01791 V=800.0 PL=0
MOVL C01792 V=800.0 PL=0
MOVL C01793 V=800.0 PL=0
MOVL C01794 V=800.0 PL=0
MOVL C01795 V=800.0 PL=0
MOVL C01796 V=800.0 PL=0
MOVL C01797 V=800.0 PL=0
MOVL C01798 V=800.0 PL=0
MOVL C01799 V=800.0 PL=0
MOVL C01800 V=800.0 PL=0
MOVL C01801 V=800.0 PL=0
MOVL C01802 V=800.0 PL=0
MOVL C01803 V=800.0 PL=0
MOVL C01804 V=800.0 PL=0
MOVL C01805 V=800.0 PL=0
MOVL C01806 V=800.0 PL=0
MOVL C01807 V=800.0 PL=0
MOVL C01808 V=800.0 PL=0
MOVL C01809 V=800.0 PL=0
MOVL C01810 V=800.0 PL=0
MOVL C01811 V=800.0 PL=0
MOVL C01812 V=800.0 PL=0
MOVL C01813 V=800.0 PL=0
MOVL C01814 V=800.0 PL=0
MOVL C01815 V=800.0 PL=0
MOVL C01816 V=800.0 PL=0
MOVL C01817 V=800.0 PL=0
MOVL C01818 V=800.0 PL=0
MOVL C01819 V=800.0 PL=0
MOVL C01820 V=800.0 PL=0
MOVL C01821 V=800.0 PL=0
MOVL C01822 V=800.0 PL=0
MOVL C01823 V=800.0 PL=0
MOVL C01824 V=800.0 PL=0
MOVL C01825 V=800.0 PL=0
MOVL C01826 V=800.0 PL=0
MOVL C01827 V=800.0 PL=0
MOVL C01828 V=800.0 PL=0
MOVL C01829 V=800.0 PL=0
MOVL C01830 V=800.0 PL=0
MOVL C01831 V=800.0 PL=0
MOVL C01832 V=800.0 PL=0
MOVL C01833 V=800.0 PL=0
MOVL C01834 V=800.0 PL=0
MOVL C01835 V=800.0 PL=0
MOVL C01836 V=800.0 PL=0
MOVL C01837 V=800.0 PL=0
MOVL C01838 V=800.0 PL=0
MOVL C01839 V=800.0 PL=0
MOVL C01840 V=800.0 PL=0
MOVL C01841 V=800.0 PL=0
MOVL C01842 V=800.0 PL=0
MOVL C01843 V=800.0 PL=0
MOVL C01844 V=800.0 PL=0
MOVL C01845 V=800.0 PL=0
MOVL C01846 V=800.0 PL=0
MOVL C01847 V=800.0 PL=0
MOVL C01848 V=800.0 PL=0
MOVL C01849 V=800.0 PL=0
MOVL C01850 V=800.0 PL=0
MOVL C01851 V=800.0 PL=0
MOVL C01852 V=800.0 PL=0
MOVL C01853 V=800.0 PL=0
MOVL C01854 V=800.0 PL=0
MOVL C01855 V=800.0 PL=0
MOVL C01856 V=800.0 PL=0
MOVL C01857 V=800.0 PL=0
MOVL C01858 V=800.0 PL=0
MOVL C01859 V=800.0 PL=0
MOVL C01860 V=800.0 PL=0
MOVL C01861 V=800.0 PL=0
MOVL C01862 V=800.0 PL=0
MOVL C01863 V=800.0 PL=0
MOVL C01864 V=800.0 PL=0
MOVL C01865 V=800.0 PL=0
MOVL C01866 V=800.0 PL=0
MOVL C01867 V=800.0 PL=0
MOVL C01868 V=800.0 PL=0
MOVL C01869 V=800.0 PL=0
MOVL C01870 V=800.0 PL=0
MOVL C01871 V=800.0 PL=0
MOVL C01872 V=800.0 PL=0
MOVL C01873 V=800.0 PL=0
MOVL C01874 V=800.0 PL=0
MOVL C01875 V=800.0 PL=0
MOVL C01876 V=800.0 PL=0
MOVL C01877 V=800.0 PL=0
MOVL C01878 V=800.0 PL=0
MOVL C01879 V=800.0 PL=0
MOVL C01880 V=800.0 PL=0
MOVL C01881 V=800.0 PL=0
MOVL C01882 V=800.0 PL=0
MOVL C01883 V=800.0 PL=0
MOVL C01884 V=800.0 PL=0
MOVL C01885 V=800.0 PL=0
MOVL C01886 V=800.0 PL=0
MOVL C01887 V=800.0 PL=0
MOVL C01888 V=800.0 PL=0
MOVL C01889 V=800.0 PL=0
MOVL C01890 V=800.0 PL=0
MOVL C01891 V=800.0 PL=0
MOVL C01892 V=800.0 PL=0
MOVL C01893 V=800.0 PL=0
MOVL C01894 V=800.0 PL=0
MOVL C01895 V=800.0 PL=0
MOVL C01896 V=800.0 PL=0
MOVL C01897 V=800.0 PL=0
MOVL C01898 V=800.0 PL=0
MOVL C01899 V=800.0 PL=0
MOVL C01900 V=800.0 PL=0
MOVL C01901 V=800.0 PL=0
MOVL C01902 V=800.0 PL=0
MOVL C01903 V=800.0 PL=0
MOVL C01904 V=800.0 PL=0
MOVL C01905 V=800.0 PL=0
MOVL C01906 V=800.0 PL=0
MOVL C01907 V=800.0 PL=0
MOVL C01908 V=800.0 PL=0
MOVL C01909 V=800.0 PL=0
MOVL C01910 V=800.0 PL=0
MOVL C01911 V=800.0 PL=0
MOVL C01912 V=800.0 PL=0
MOVL C01913 V=800.0 PL=0
MOVL C01914 V=800.0 PL=0
MOVL C01915 V=800.0 PL=0
MOVL C01916 V=800.0 PL=0
MOVL C01917 V=800.0 PL=0
MOVL C01918 V=800.0 PL=0
MOVL C01919 V=800.0 PL=0
MOVL C01920 V=800.0 PL=0
MOVL C01921 V=800.0 PL=0
MOVL C01922 V=800.0 PL=0
MOVL C01923 V=800.0 PL=0
MOVL C01924 V=800.0 PL=0
MOVL C01925 V=800.0 PL=0
MOVL C01926 V=800.0 PL=0
MOVL C01927 V=800.0 PL=0
MOVL C01928 V=800.0 PL=0
MOVL C01929 V=800.0 PL=0
MOVL C01930 V=800.0 PL=0
MOVL C01931 V=800.0 PL=0
MOVL C01932 V=800.0 PL=0
MOVL C01933 V=800.0 PL=0
MOVL C01934 V=800.0 PL=0
MOVL C01935 V=800.0 PL=0
MOVL C01936 V=800.0 PL=0
MOVL C01937 V=800.0 PL=0
MOVL C01938 V=800.0 PL=0
MOVL C01939 V=800.0 PL=0
MOVL C01940 V=800.0 PL=0
MOVL C01941 V=800.0 PL=0
MOVL C01942 V=800.0 PL=0
MOVL C01943 V=800.0 PL=0
MOVL C01944 V=800.0 PL=0
MOVL C01945 V=800.0 PL=0
MOVL C01946 V=800.0 PL=0
MOVL C01947 V=800.0 PL=0
MOVL C01948 V=800.0 PL=0
MOVL C01949 V=800.0 PL=0
MOVL C01950 V=800.0 PL=0
MOVL C01951 V=800.0 PL=0
MOVL C01952 V=800.0 PL=0
MOVL C01953 V=800.0 PL=0
MOVL C01954 V=800.0 PL=0
MOVL C01955 V=800.0 PL=0
MOVL C01956 V=800.0 PL=0
MOVL C01957 V=800.0 PL=0
MOVL C01958 V=800.0 PL=0
MOVL C01959 V=800.0 PL=0
MOVL C01960 V=800.0 PL=0
MOVL C01961 V=800.0 PL=0
MOVL C01962 V=800.0 PL=0
MOVL C01963 V=800.0 PL=0
MOVL C01964 V=800.0 PL=0
MOVL C01965 V=800.0 PL=0
MOVL C01966 V=800.0 PL=0
MOVL C01967 V=800.0 PL=0
MOVL C01968 V=800.0 PL=0
MOVL C01969 V=800.0 PL=0
MOVL C01970 V=800.0 PL=0
MOVL C01971 V=800.0 PL=0
MOVL C01972 V=800.0 PL=0
MOVL C01973 V=800.0 PL=0
MOVL C01974 V=800.0 PL=0
MOVL C01975 V=800.0 PL=0
MOVL C01976 V=800.0 PL=0
MOVL C01977 V=800.0 PL=0
MOVL C01978 V=800.0 PL=0
MOVL C01979 V=800.0 PL=0
MOVL C01980 V=800.0 PL=0
MOVL C01981 V=800.0 PL=0
MOVL C01982 V=800.0 PL=0
MOVL C01983 V=800.0 PL=0
MOVL C01984 V=800.0 PL=0
MOVL C01985 V=800.0 PL=0
MOVL C01986 V=800.0 PL=0
MOVL C01987 V=800.0 PL=0
MOVL C01988 V=800.0 PL=0
MOVL C01989 V=800.0 PL=0
MOVL C01990 V=800.0 PL=0
MOVL C01991 V=800.0 PL=0
MOVL C01992 V=800.0 PL=0
MOVL C01993 V=800.0 PL=0
MOVL C01994 V=800.0 PL=0
MOVL C01995 V=800.0 PL=0
MOVL C01996 V=800.0 PL=0
MOVL C01997 V=800.0 PL=0
MOVL C01998 V=800.0 PL=0
MOVL C01999 V=800.0 PL=0
MOVL C02000 V=800.0 PL=0
MOVL C02001 V=800.0 PL=0
MOVL C02002 V=800.0 PL=0
MOVL C02003 V=800.0 PL=0
MOVL C02004 V=800.0 PL=0
MOVL C02005 V=800.0 PL=0
MOVL C02006 V=800.0 PL=0
MOVL C02007 V=800.0 PL=0
MOVL C02008 V=800.0 PL=0
MOVL C02009 V=800.0 PL=0
MOVL C02010 V=800.0 PL=0
MOVL C02011 V=800.0 PL=0
MOVL C02012 V=800.0 PL=0
MOVL C02013 V=800.0 PL=0
MOVL C02014 V=800.0 PL=0
MOVL C02015 V=800.0 PL=0
MOVL C02016 V=800.0 PL=0
MOVL C02017 V=800.0 PL=0
MOVL C02018 V=800.0 PL=0
MOVL C02019 V=800.0 PL=0
MOVL C02020 V=800.0 PL=0
MOVL C02021 V=800.0 PL=0
MOVL C02022 V=800.0 PL=0
MOVL C02023 V=800.0 PL=0
MOVL C02024 V=800.0 PL=0
MOVL C02025 V=800.0 PL=0
MOVL C02026 V=800.0 PL=0
MOVL C02027 V=800.0 PL=0
MOVL C02028 V=800.0 PL=0
MOVL C02029 V=800.0 PL=0
MOVL C02030 V=800.0 PL=0
MOVL C02031 V=800.0 PL=0
MOVL C02032 V=800.0 PL=0
MOVL C02033 V=800.0 PL=0
MOVL C02034 V=800.0 PL=0
MOVL C02035 V=800.0 PL=0
MOVL C02036 V=800.0 PL=0
MOVL C02037 V=800.0 PL=0
MOVL C02038 V=800.0 PL=0
MOVL C02039 V=800.0 PL=0
MOVL C02040 V=800.0 PL=0
MOVL C02041 V=800.0 PL=0
MOVL C02042 V=800.0 PL=0
MOVL C02043 V=800.0 PL=0
MOVL C02044 V=800.0 PL=0
MOVL C02045 V=800.0 PL=0
MOVL C02046 V=800.0 PL=0
MOVL C02047 V=800.0 PL=0
MOVL C02048 V=800.0 PL=0
MOVL C02049 V=800.0 PL=0
MOVL C02050 V=800.0 PL=0
MOVL C02051 V=800.0 PL=0
MOVL C02052 V=800.0 PL=0
MOVL C02053 V=800.0 PL=0
MOVL C02054 V=800.0 PL=0
MOVL C02055 V=800.0 PL=0
MOVL C02056 V=800.0 PL=0
MOVL C02057 V=800.0 PL=0
MOVL C02058 V=800.0 PL=0
MOVL C02059 V=800.0 PL=0
MOVL C02060 V=800.0 PL=0
MOVL C02061 V=800.0 PL=0
MOVL C02062 V=800.0 PL=0
MOVL C02063 V=800.0 PL=0
MOVL C02064 V=800.0 PL=0
MOVL C02065 V=800.0 PL=0
MOVL C02066 V=800.0 PL=0
MOVL C02067 V=800.0 PL=0
MOVL C02068 V=800.0 PL=0
MOVL C02069 V=800.0 PL=0
MOVL C02070 V=800.0 PL=0
MOVL C02071 V=800.0 PL=0
MOVL C02072 V=800.0 PL=0
MOVL C02073 V=800.0 PL=0
MOVL C02074 V=800.0 PL=0
MOVL C02075 V=800.0 PL=0
MOVL C02076 V=800.0 PL=0
MOVL C02077 V=800.0 PL=0
MOVL C02078 V=800.0 PL=0
MOVL C02079 V=800.0 PL=0
MOVL C02080 V=800.0 PL=0
MOVL C02081 V=800.0 PL=0
MOVL C02082 V=800.0 PL=0
MOVL C02083 V=800.0 PL=0
MOVL C02084 V=800.0 PL=0
MOVL C02085 V=800.0 PL=0
MOVL C02086 V=800.0 PL=0
MOVL C02087 V=800.0 PL=0
MOVL C02088 V=800.0 PL=0
MOVL C02089 V=800.0 PL=0
MOVL C02090 V=800.0 PL=0
MOVL C02091 V=800.0 PL=0
MOVL C02092 V=800.0 PL=0
MOVL C02093 V=800.0 PL=0
MOVL C02094 V=800.0 PL=0
MOVL C02095 V=800.0 PL=0
MOVL C02096 V=800.0 PL=0
MOVL C02097 V=800.0 PL=0
MOVL C02098 V=800.0 PL=0
MOVL C02099 V=800.0 PL=0
MOVL C02100 V=800.0 PL=0
MOVL C02101 V=800.0 PL=0
MOVL C02102 V=800.0 PL=0
MOVL C02103 V=800.0 PL=0
MOVL C02104 V=800.0 PL=0
MOVL C02105 V=800.0 PL=0
MOVL C02106 V=800.0 PL=0
MOVL C02107 V=800.0 PL=0
MOVL C02108 V=800.0 PL=0
MOVL C02109 V=800.0 PL=0
MOVL C02110 V=800.0 PL=0
MOVL C02111 V=800.0 PL=0
MOVL C02112 V=800.0 PL=0
MOVL C02113 V=800.0 PL=0
MOVL C02114 V=800.0 PL=0
MOVL C02115 V=800.0 PL=0
MOVL C02116 V=800.0 PL=0
MOVL C02117 V=800.0 PL=0
MOVL C02118 V=800.0 PL=0
MOVL C02119 V=800.0 PL=0
MOVL C02120 V=800.0 PL=0
MOVL C02121 V=800.0 PL=0
MOVL C02122 V=800.0 PL=0
MOVL C02123 V=800.0 PL=0
MOVL C02124 V=800.0 PL=0
MOVL C02125 V=800.0 PL=0
MOVL C02126 V=800.0 PL=0
MOVL C02127 V=800.0 PL=0
MOVL C02128 V=800.0 PL=0
MOVL C02129 V=800.0 PL=0
MOVL C02130 V=800.0 PL=0
MOVL C02131 V=800.0 PL=0
MOVL C02132 V=800.0 PL=0
MOVL C02133 V=800.0 PL=0
MOVL C02134 V=800.0 PL=0
MOVL C02135 V=800.0 PL=0
MOVL C02136 V=800.0 PL=0
MOVL C02137 V=800.0 PL=0
MOVL C02138 V=800.0 PL=0
MOVL C02139 V=800.0 PL=0
MOVL C02140 V=800.0 PL=0
MOVL C02141 V=800.0 PL=0
MOVL C02142 V=800.0 PL=0
MOVL C02143 V=800.0 PL=0
MOVL C02144 V=800.0 PL=0
MOVL C02145 V=800.0 PL=0
MOVL C02146 V=800.0 PL=0
MOVL C02147 V=800.0 PL=0
MOVL C02148 V=800.0 PL=0
MOVL C02149 V=800.0 PL=0
MOVL C02150 V=800.0 PL=0
MOVL C02151 V=800.0 PL=0
MOVL C02152 V=800.0 PL=0
MOVL C02153 V=800.0 PL=0
MOVL C02154 V=800.0 PL=0
MOVL C02155 V=800.0 PL=0
MOVL C02156 V=800.0 PL=0
MOVL C02157 V=800.0 PL=0
MOVL C02158 V=800.0 PL=0
MOVL C02159 V=800.0 PL=0
MOVL C02160 V=800.0 PL=0
MOVL C02161 V=800.0 PL=0
MOVL C02162 V=800.0 PL=0
MOVL C02163 V=800.0 PL=0
MOVL C02164 V=800.0 PL=0
MOVL C02165 V=800.0 PL=0
